(*Call actual FBs*)
fb_Move_ABS[Axis_Index](Axis:= Axis[Axis_Index]);
IF ReadyFor_Motion[Axis_Index] AND In_Play_ACK[Axis_Index] AND NOT FB_In.Stop_PlayBack[Axis_Index] AND NOT Cycle_Complete[Axis_Index]
	THEN
			(*---------------Explicit Step Call-------------*)
			IF (FB_In.Start_Explicit_StepCall[Axis_Index] OR Step_Running[Axis_Index])
				AND (NOT FB_In.Start_PlayBack[Axis_Index] OR Step_Running[Axis_Index]) AND NOT Program_Running[Axis_Index]
				AND NOT Step_Complete[Axis_Index]
				AND (Current_Step_Pointer[Axis_Index]>=1) AND (Current_Step_Pointer[Axis_Index]<=15)
					THEN
					Step_Running[Axis_Index]:= TRUE;
					Current_Step_Pointer[Axis_Index]:= FB_In.Explicit_Step_REQ[Axis_Index];
					(*--- Absolute Type Move Requested ---*)
					IF NOT fb_Move_ABS[Axis_Index].Active AND NOT fb_Move_Vel[Axis_Index].Active AND NOT fb_Move_MOD[Axis_Index].Active
						AND NOT fb_Move_ABS[Axis_Index].Execute AND NOT fb_Move_Vel[Axis_Index].Execute AND NOT fb_Move_MOD[Axis_Index].Execute
						AND (Program_Positions[Axis_Index][Current_Step_Pointer[Axis_Index]].Move_Type=0)
						THEN
						(*Set Auto Playback Parameters Per Position*)
						fb_Move_ABS[Axis_Index].Velocity:= (Program_Positions[Axis_Index] [Current_Step_Pointer[Axis_Index]].Velocity *(FB_In.PlayBack_Speed_Percentage[Axis_Index]/100));
						fb_Move_ABS[Axis_Index].Acceleration:= Program_Positions[Axis_Index][Current_Step_Pointer[Axis_Index]].Accel;
						fb_Move_ABS[Axis_Index].Deceleration:= Program_Positions[Axis_Index][Current_Step_Pointer[Axis_Index]].Decel;
						fb_Move_ABS[Axis_Index].Position:= Program_Positions[Axis_Index][Current_Step_Pointer[Axis_Index]].Position;
						fb_Move_ABS[Axis_Index].Execute:= TRUE;
					ELSIF fb_Move_ABS[Axis_Index].Execute AND fb_Move_ABS[Axis_Index].Done AND In_Requested_Position[Axis_Index] AND (At_Current_Step[Axis_Index] = Current_Step_Pointer[Axis_Index])
						THEN
							fb_Move_ABS[Axis_Index].Execute:= FALSE;			(*Position Reached, step execution request*)
							Step_Complete[Axis_Index]:= TRUE;
					END_IF;

			END_IF;

			(*--------------Cycle through Programmed Steps Continuous until End-----------*)
			IF (FB_In.Start_PlayBack[Axis_Index])
				AND fb_Power[Axis_Index].Status (*MC_Power -> Status:=Control Loop Closed (new ready bit (StateDWord.20) and not in error*)
				AND NOT FB_In.Start_Explicit_StepCall[Axis_Index] AND NOT Step_Running[Axis_Index]
				AND NOT Program_Complete[Axis_Index] AND FB_In.PlayBack_StepPermit[Axis_Index]
				AND ((NOT Program_Running[Axis_Index] AND ((Current_Step_Pointer[Axis_Index]=1) AND In_Requested_Position[Axis_Index]))
				OR (Program_Running[Axis_Index] AND (Current_Step_Pointer[Axis_Index]>=1) AND (Current_Step_Pointer[Axis_Index]<=15)))
					THEN
					Program_Running[Axis_Index]:= TRUE;
					IF NOT fb_Move_ABS[Axis_Index].Active AND NOT fb_Move_ABS[Axis_Index].Execute
						AND NOT fb_Move_MOD[Axis_Index].Active AND NOT fb_Move_MOD[Axis_Index].Execute
						AND (Program_Positions[Axis_Index][Current_Step_Pointer[Axis_Index]].Move_Type=0)
						THEN
						(*Set Auto Playback Parameters Per Position*)
						fb_Move_ABS[Axis_Index].Velocity:= (Program_Positions[Axis_Index][Current_Step_Pointer[Axis_Index]].Velocity *(FB_In.PlayBack_Speed_Percentage[Axis_Index]/100));
						fb_Move_ABS[Axis_Index].Acceleration:= Program_Positions[Axis_Index][Current_Step_Pointer[Axis_Index]].Accel;
						fb_Move_ABS[Axis_Index].Deceleration:= Program_Positions[Axis_Index][Current_Step_Pointer[Axis_Index]].Decel;
						fb_Move_ABS[Axis_Index].Position:= Program_Positions[Axis_Index][Current_Step_Pointer[Axis_Index]].Position;
						fb_Move_ABS[Axis_Index].Execute:= TRUE;
					ELSIF fb_Move_ABS[Axis_Index].Execute AND fb_Move_ABS[Axis_Index].Done AND In_Requested_Position[Axis_Index] AND (At_Current_Step[Axis_Index] = Current_Step_Pointer[Axis_Index])
						THEN
							fb_Move_ABS[Axis_Index].Execute:= FALSE; 				(*Position Reached, step execution request*)
							(*Set Program Complete Flag to Only Allow One Cycle*)
							IF Program_Running[Axis_Index] AND Current_Step_Pointer[Axis_Index]> 15 OR (Program_Positions[Axis_Index][Current_Step_Pointer[Axis_Index]].End_Flag=TRUE)
								THEN
									Program_Complete[Axis_Index]:= TRUE;
							END_IF;
							Current_Step_Pointer[Axis_Index]:= Current_Step_Pointer[Axis_Index]+1;	(*Once Position is reached, increment step pointer*)
					END_IF;
			END_IF;

(*Call actual FBs*)
fb_Move_ABS[Axis_Index](Axis:= Axis[Axis_Index]);

				(*Reset Complete Flag and Step Pointer*)
				IF (Program_Complete[Axis_Index] AND Program_Running[Axis_Index]) OR FB_In.Program_Reset[Axis_Index]
					THEN
						Current_Step_Pointer[Axis_Index]:= 1;
						IF NOT fb_Move_ABS[Axis_Index].Busy AND NOT fb_Move_ABS[Axis_Index].Execute
							AND NOT fb_Move_MOD[Axis_Index].Busy AND NOT fb_Move_MOD[Axis_Index].Execute
							THEN
							(*Set Auto Playback Parameters Per Position*)
							fb_Move_ABS[Axis_Index].Velocity:= (Program_Positions[Axis_Index][Current_Step_Pointer[Axis_Index]].Velocity *(FB_In.PlayBack_Speed_Percentage[Axis_Index]/100));
							fb_Move_ABS[Axis_Index].Acceleration:= Program_Positions[Axis_Index][Current_Step_Pointer[Axis_Index]].Accel;
							fb_Move_ABS[Axis_Index].Deceleration:= Program_Positions[Axis_Index][Current_Step_Pointer[Axis_Index]].Decel;
							fb_Move_ABS[Axis_Index].Position:= Program_Positions[Axis_Index][Current_Step_Pointer[Axis_Index]].Position;
							fb_Move_ABS[Axis_Index].Execute:= TRUE;
						ELSIF fb_Move_ABS[Axis_Index].Execute AND fb_Move_ABS[Axis_Index].Done AND In_Requested_Position[Axis_Index] AND (At_Current_Step[Axis_Index] = Current_Step_Pointer[Axis_Index])
							THEN
								fb_Move_ABS[Axis_Index].Execute:= FALSE; 				(*Position Reached, step execution request*)
								Program_Complete[Axis_Index]:= FALSE;
								Program_Running[Axis_Index]:= FALSE;
								Cycle_Complete[Axis_Index]:= TRUE;
						END_IF;
				END_IF;



ELSE
	fb_Move_ABS[Axis_Index].Execute:= FALSE;
	fb_Move_VEL[Axis_Index].Execute:= FALSE;
	fb_Move_MOD[Axis_Index].Execute:= FALSE;
	Step_Complete[Axis_Index]:= FALSE;
	Step_Running[Axis_Index]:= FALSE;

END_IF; (*End_If for Play Loop*)
END_ACTION

ACTION Move_Modulo:
(*General Set-Up Parameters/Function calls for Servo Drive*)

(*Call actual FBs*)
fb_Move_MOD[Axis_Index](Axis:= Axis[Axis_Index]);
IF ReadyFor_Motion[Axis_Index] AND In_Play_ACK[Axis_Index] AND NOT FB_In.Stop_PlayBack[Axis_Index] AND NOT Cycle_Complete[Axis_Index]
	THEN
			(*---------------Explicit Step Call-------------*)
			IF (FB_In.Start_Explicit_StepCall[Axis_Index] OR Step_Running[Axis_Index])
				AND (NOT FB_In.Start_PlayBack[Axis_Index] OR Step_Running[Axis_Index]) AND NOT Program_Running[Axis_Index]
				AND NOT Step_Complete[Axis_Index]
				AND (Current_Step_Pointer[Axis_Index]>=1) AND (Current_Step_Pointer[Axis_Index]<=15)
					THEN
					Step_Running[Axis_Index]:= TRUE;
					Current_Step_Pointer[Axis_Index]:= FB_In.Explicit_Step_REQ[Axis_Index];
					(*--- Modulo Type Move Requested ---*)
					IF NOT fb_Move_ABS[Axis_Index].Active AND NOT fb_Move_Vel[Axis_Index].Active AND NOT fb_Move_MOD[Axis_Index].Active
						AND NOT fb_Move_ABS[Axis_Index].Execute AND NOT fb_Move_Vel[Axis_Index].Execute AND NOT fb_Move_MOD[Axis_Index].Execute
						AND (Program_Positions[Axis_Index][Current_Step_Pointer[Axis_Index]].Move_Type=3)
						THEN
						(*Set Auto Playback Parameters Per Position*)
						fb_Move_MOD[Axis_Index].Velocity:= (Program_Positions[Axis_Index] [Current_Step_Pointer[Axis_Index]].Velocity *(FB_In.PlayBack_Speed_Percentage[Axis_Index]/100));
						fb_Move_MOD[Axis_Index].Acceleration:= Program_Positions[Axis_Index][Current_Step_Pointer[Axis_Index]].Accel;
						fb_Move_MOD[Axis_Index].Deceleration:= Program_Positions[Axis_Index][Current_Step_Pointer[Axis_Index]].Decel;
						fb_Move_MOD[Axis_Index].Position:= Program_Positions[Axis_Index][Current_Step_Pointer[Axis_Index]].Position;
						fb_Move_MOD[Axis_Index].Execute:= TRUE;
					ELSIF fb_Move_MOD[Axis_Index].Execute AND fb_Move_MOD[Axis_Index].Done AND In_Requested_Position[Axis_Index] AND (At_Current_Step[Axis_Index] = Current_Step_Pointer[Axis_Index])
						THEN
							fb_Move_MOD[Axis_Index].Execute:= FALSE;			(*Position Reached, step execution request*)
							Step_Complete[Axis_Index]:= TRUE;
					END_IF;

			END_IF;

			(*--------------Cycle through Programmed Steps Continuous until End-----------*)
			IF (FB_In.Start_PlayBack[Axis_Index])
				AND fb_Power[Axis_Index].Status (*MC_Power -> Status:=Control Loop Closed (new ready bit (StateDWord.20) and not in error*)
				AND NOT FB_In.Start_Explicit_StepCall[Axis_Index] AND NOT Step_Running[Axis_Index]
				AND NOT Program_Complete[Axis_Index] AND FB_In.PlayBack_StepPermit[Axis_Index]
				AND ((NOT Program_Running[Axis_Index] AND ((Current_Step_Pointer[Axis_Index]=1) AND In_Requested_Position[Axis_Index]))
				OR (Program_Running[Axis_Index] AND (Current_Step_Pointer[Axis_Index]>=1) AND (Current_Step_Pointer[Axis_Index]<=15)))
					THEN
					Program_Running[Axis_Index]:= TRUE;
					IF NOT fb_Move_ABS[Axis_Index].Active AND NOT fb_Move_ABS[Axis_Index].Execute
						AND NOT fb_Move_MOD[Axis_Index].Active AND NOT fb_Move_MOD[Axis_Index].Execute
						AND (Program_Positions[Axis_Index][Current_Step_Pointer[Axis_Index]].Move_Type=0)
						THEN
						(*Set Auto Playback Parameters Per Position*)
						fb_Move_MOD[Axis_Index].Velocity:= (Program_Positions[Axis_Index][Current_Step_Pointer[Axis_Index]].Velocity *(FB_In.PlayBack_Speed_Percentage[Axis_Index]/100));
						fb_Move_MOD[Axis_Index].Acceleration:= Program_Positions[Axis_Index][Current_Step_Pointer[Axis_Index]].Accel;
						fb_Move_MOD[Axis_Index].Deceleration:= Program_Positions[Axis_Index][Current_Step_Pointer[Axis_Index]].Decel;
						fb_Move_MOD[Axis_Index].Position:= Program_Positions[Axis_Index][Current_Step_Pointer[Axis_Index]].Position;
						fb_Move_MOD[Axis_Index].Execute:= TRUE;
					ELSIF fb_Move_MOD[Axis_Index].Execute AND fb_Move_MOD[Axis_Index].Done AND In_Requested_Position[Axis_Index] AND (At_Current_Step[Axis_Index] = Current_Step_Pointer[Axis_Index])
						THEN
							fb_Move_MOD[Axis_Index].Execute:= FALSE; 				(*Position Reached, step execution request*)
							(*Set Program Complete Flag to Only Allow One Cycle*)
							IF Program_Running[Axis_Index] AND Current_Step_Pointer[Axis_Index]> 15 OR (Program_Positions[Axis_Index][Current_Step_Pointer[Axis_Index]].End_Flag=TRUE)
								THEN
									Program_Complete[Axis_Index]:= TRUE;
							END_IF;
							Current_Step_Pointer[Axis_Index]:= Current_Step_Pointer[Axis_Index]+1;	(*Once Position is reached, increment step pointer*)
					END_IF;
			END_IF;

(*Call actual FBs*)
fb_Move_MOD[Axis_Index](Axis:= Axis[Axis_Index]);

				(*Reset Complete Flag and Step Pointer*)
				IF (Program_Complete[Axis_Index] AND Program_Running[Axis_Index]) OR FB_In.Program_Reset[Axis_Index]
					THEN
						Current_Step_Pointer[Axis_Index]:= 1;
						IF NOT fb_Move_ABS[Axis_Index].Busy AND NOT fb_Move_ABS[Axis_Index].Execute
							AND NOT fb_Move_MOD[Axis_Index].Busy AND NOT fb_Move_MOD[Axis_Index].Execute
							THEN
							(*Set Auto Playback Parameters Per Position*)
							fb_Move_MOD[Axis_Index].Velocity:= (Program_Positions[Axis_Index][Current_Step_Pointer[Axis_Index]].Velocity *(FB_In.PlayBack_Speed_Percentage[Axis_Index]/100));
							fb_Move_MOD[Axis_Index].Acceleration:= Program_Positions[Axis_Index][Current_Step_Pointer[Axis_Index]].Accel;
							fb_Move_MOD[Axis_Index].Deceleration:= Program_Positions[Axis_Index][Current_Step_Pointer[Axis_Index]].Decel;
							fb_Move_MOD[Axis_Index].Position:= Program_Positions[Axis_Index][Current_Step_Pointer[Axis_Index]].Position;
							fb_Move_MOD[Axis_Index].Execute:= TRUE;
						ELSIF fb_Move_MOD[Axis_Index].Execute AND fb_Move_MOD[Axis_Index].Done AND In_Requested_Position[Axis_Index] AND (At_Current_Step[Axis_Index] = Current_Step_Pointer[Axis_Index])
							THEN
								fb_Move_MOD[Axis_Index].Execute:= FALSE; 				(*Position Reached, step execution request*)
								Program_Complete[Axis_Index]:= FALSE;
								Program_Running[Axis_Index]:= FALSE;
								Cycle_Complete[Axis_Index]:= TRUE;
						END_IF;
				END_IF;



ELSE
	fb_Move_ABS[Axis_Index].Execute:= FALSE;
	fb_Move_VEL[Axis_Index].Execute:= FALSE;
	fb_Move_MOD[Axis_Index].Execute:= FALSE;
	Step_Complete[Axis_Index]:= FALSE;
	Step_Running[Axis_Index]:= FALSE;

END_IF; (*End_If for Play Loop*)
END_ACTION

ACTION Move_Velocity:
(*General Set-Up Parameters/Function calls for Servo Drive*)

(*Call actual FBs*)
fb_Move_Vel[Axis_Index](Axis:= Axis[Axis_Index]);

IF ReadyFor_Motion[Axis_Index] AND In_Play_ACK[Axis_Index] AND NOT FB_In.Stop_PlayBack[Axis_Index] AND NOT Cycle_Complete[Axis_Index]
	THEN
			(*---------------Explicit Step Call-------------*)
			IF (FB_In.Start_Explicit_StepCall[Axis_Index] OR Step_Running[Axis_Index])
				AND (NOT FB_In.Start_PlayBack[Axis_Index] OR Step_Running[Axis_Index]) AND NOT Program_Running[Axis_Index]
				AND NOT Step_Complete[Axis_Index]
				AND (Current_Step_Pointer[Axis_Index]>=1) AND (Current_Step_Pointer[Axis_Index]<=15)
					THEN
					Step_Running[Axis_Index]:= TRUE;
					Current_Step_Pointer[Axis_Index]:= FB_In.Explicit_Step_REQ[Axis_Index];

					(*--- Velocity only type move requested (+ or - direction) ---*)
					IF NOT fb_Move_ABS[Axis_Index].Active AND NOT fb_Move_Vel[Axis_Index].Active AND NOT fb_Move_MOD[Axis_Index].Active
						AND NOT fb_Move_ABS[Axis_Index].Execute AND NOT fb_Move_Vel[Axis_Index].Execute AND NOT fb_Move_MOD[Axis_Index].Execute
						AND ((Program_Positions[Axis_Index][Current_Step_Pointer[Axis_Index]].Move_Type=1) OR  (Program_Positions[Axis_Index][Current_Step_Pointer[Axis_Index]].Move_Type=2))

						THEN
						(*Set Auto Playback Parameters Per Position*)
						fb_Move_VEL[Axis_Index].Velocity:= (Program_Positions[Axis_Index] [Current_Step_Pointer[Axis_Index]].Velocity *(FB_In.PlayBack_Speed_Percentage[Axis_Index]/100));
						fb_Move_VEL[Axis_Index].Acceleration:= Program_Positions[Axis_Index][Current_Step_Pointer[Axis_Index]].Accel;
						fb_Move_VEL[Axis_Index].Deceleration:= Program_Positions[Axis_Index][Current_Step_Pointer[Axis_Index]].Decel;
						(*Set Directionality*)
						IF (Program_Positions[Axis_Index][Current_Step_Pointer[Axis_Index]].Move_Type=1) (*+ direction requested*)
							THEN
							fb_Move_VEL[Axis_Index].Direction:= MC_Positive_Direction; (*Set Direction to Positive*)
						ELSIF (Program_Positions[Axis_Index][Current_Step_Pointer[Axis_Index]].Move_Type=2) (*- direction requested*)
							THEN
							fb_Move_VEL[Axis_Index].Direction:= MC_Negative_Direction; (*Set Direction to Positive*)
						END_IF;
						fb_Move_VEL[Axis_Index].Execute:= TRUE;
					END_IF;
			END_IF;

ELSE
	fb_Move_ABS[Axis_Index].Execute:= FALSE;
	fb_Move_VEL[Axis_Index].Execute:= FALSE;
	fb_Move_MOD[Axis_Index].Execute:= FALSE;
	Step_Complete[Axis_Index]:= FALSE;
	Step_Running[Axis_Index]:= FALSE;

END_IF; (*End_If for Play Loop*)
END_ACTION

ACTION Teach_Mode:
(*################################################# Manual Mode Code ###########################################*)
(*General Set-Up Parameters/Function calls for Servo Drive*)
			fb_Jog[Axis_Index](Axis:= Axis[Axis_Index]);
			fb_Move_ABSTeach[Axis_Index](Axis:= Axis[Axis_Index]);
			fb_Set_Home[Axis_Index](Axis:= Axis[Axis_Index]);
			SET_HomeTMR[Axis_Index].PT:= T#5.0s;							(*Preset Time for Teach HomePos*)

IF ReadyFor_TeachMotion[Axis_Index] AND In_Teach_ACK[Axis_Index] AND NOT fb_Stop[Axis_Index].Execute
	THEN
		Current_Step_Pointer[Axis_Index]:= FB_In.Explicit_Step_REQ[Axis_Index];
		Step_Complete[Axis_Index]:= FALSE;
		Step_Running[Axis_Index]:= FALSE;
		Program_Complete[Axis_Index]:= FALSE;
		Program_Running[Axis_Index]:= FALSE;

			(*---------------Explicit Step Call in Teach-------------*)
			IF FB_In.Start_Explicit_StepCall[Axis_Index] AND ReadyFor_Motion[Axis_Index]
				AND (Current_Step_Pointer[Axis_Index]>=1) AND (Current_Step_Pointer[Axis_Index]<=15)
					THEN
					(*--- Absolute Type Move Requested ---*)
					IF NOT fb_Move_ABS[Axis_Index].Active AND NOT fb_Move_Vel[Axis_Index].Active AND NOT fb_Move_MOD[Axis_Index].Active
						AND NOT fb_Move_ABS[Axis_Index].Execute AND NOT fb_Move_Vel[Axis_Index].Execute AND NOT fb_Move_MOD[Axis_Index].Execute
						AND (Program_Positions[Axis_Index][Current_Step_Pointer[Axis_Index]].Move_Type=0)
						THEN
						(*Set Auto Playback Parameters Per Position*)
						fb_Move_ABS[Axis_Index].Velocity:= 250; (*In Teach Mode, Lock down Velcoity*)
						fb_Move_ABS[Axis_Index].Acceleration:= Program_Positions[Axis_Index][Current_Step_Pointer[Axis_Index]].Accel;
						fb_Move_ABS[Axis_Index].Deceleration:= Program_Positions[Axis_Index][Current_Step_Pointer[Axis_Index]].Decel;
						fb_Move_ABS[Axis_Index].Position:= Program_Positions[Axis_Index][Current_Step_Pointer[Axis_Index]].Position;
						fb_Move_ABS[Axis_Index].Execute:= TRUE;
					ELSIF fb_Move_ABS[Axis_Index].Execute AND fb_Move_ABS[Axis_Index].Done AND In_Requested_Position[Axis_Index] AND (At_Current_Step[Axis_Index] = Current_Step_Pointer[Axis_Index])
						THEN
							fb_Move_ABS[Axis_Index].Execute:= FALSE;			(*Position Reached, step execution request*)
					END_IF;
					(*--- Modulo Type Move Requested ---*)
					IF NOT fb_Move_ABS[Axis_Index].Active AND NOT fb_Move_Vel[Axis_Index].Active AND NOT fb_Move_MOD[Axis_Index].Active
						AND NOT fb_Move_ABS[Axis_Index].Execute AND NOT fb_Move_Vel[Axis_Index].Execute AND NOT fb_Move_MOD[Axis_Index].Execute
						AND (Program_Positions[Axis_Index][Current_Step_Pointer[Axis_Index]].Move_Type=3)
						THEN
						(*Set Auto Playback Parameters Per Position*)
						fb_Move_MOD[Axis_Index].Velocity:= 250; (*In Teach Mode, Lock down Velcoity*)
						fb_Move_MOD[Axis_Index].Acceleration:= Program_Positions[Axis_Index][Current_Step_Pointer[Axis_Index]].Accel;
						fb_Move_MOD[Axis_Index].Deceleration:= Program_Positions[Axis_Index][Current_Step_Pointer[Axis_Index]].Decel;
						fb_Move_MOD[Axis_Index].Position:= Program_Positions[Axis_Index][Current_Step_Pointer[Axis_Index]].Position;
						fb_Move_MOD[Axis_Index].Execute:= TRUE;
					ELSIF fb_Move_MOD[Axis_Index].Execute AND fb_Move_MOD[Axis_Index].Done AND In_Requested_Position[Axis_Index] AND (At_Current_Step[Axis_Index] = Current_Step_Pointer[Axis_Index])
						THEN
							fb_Move_MOD[Axis_Index].Execute:= FALSE;			(*Position Reached, step execution request*)
					END_IF;
					(*--- Velocity only type move requested (+ or - direction) ---*)
					IF NOT fb_Move_ABS[Axis_Index].Active AND NOT fb_Move_Vel[Axis_Index].Active
						AND NOT fb_Move_ABS[Axis_Index].Execute AND NOT fb_Move_Vel[Axis_Index].Execute
						AND ((Program_Positions[Axis_Index][Current_Step_Pointer[Axis_Index]].Move_Type=1) OR  (Program_Positions[Axis_Index][Current_Step_Pointer[Axis_Index]].Move_Type=2))
						THEN
						(*Set Auto Playback Parameters Per Position*)
						fb_Move_VEL[Axis_Index].Velocity:= 250; (*In Teach Mode, Lock down Velcoity*)
						fb_Move_VEL[Axis_Index].Acceleration:= Program_Positions[Axis_Index][Current_Step_Pointer[Axis_Index]].Accel;
						fb_Move_VEL[Axis_Index].Deceleration:= Program_Positions[Axis_Index][Current_Step_Pointer[Axis_Index]].Decel;
						(*Set Directionality*)
						IF (Program_Positions[Axis_Index][Current_Step_Pointer[Axis_Index]].Move_Type=1) (*+ direction requested*)
							THEN
							fb_Move_VEL[Axis_Index].Direction:= MC_Positive_Direction; (*Set Direction to Positive*)
						ELSIF (Program_Positions[Axis_Index][Current_Step_Pointer[Axis_Index]].Move_Type=2) (*- direction requested*)
							THEN
							fb_Move_VEL[Axis_Index].Direction:= MC_Negative_Direction; (*Set Direction to Positive*)
						END_IF;
						fb_Move_VEL[Axis_Index].Execute:= TRUE;
					END_IF;
			ELSE
				fb_Move_ABS[Axis_Index].Execute:= FALSE;
				fb_Move_VEL[Axis_Index].Execute:= FALSE;
				fb_Move_MOD[Axis_Index].Execute:= FALSE;
			END_IF;
(*Call actual FBs*)
fb_Move_ABS[Axis_Index](Axis:= Axis[Axis_Index]);
fb_Move_Vel[Axis_Index](Axis:= Axis[Axis_Index]);
fb_Move_MOD[Axis_Index](Axis:= Axis[Axis_Index]);
			(*Set Inching Value*)
			IF FB_In.Teach_MicroInch_Enable[Axis_Index]
				THEN
				Inching_Value[Axis_Index]:= FB_In.MicroInch_Value[Axis_Index];
			ELSE
				Inching_Value[Axis_Index]:= 0.5;	(*Default Inching Value is 0.5mm OR degrees (depending on how Motion System is config'd*)
			END_IF;
			(*-------------Jog and Inching -----------------------*)
			IF FB_In.Teach_JogFast_Plus[Axis_Index] OR FB_In.Teach_JogFast_Minus[Axis_Index]
				THEN
					(*Jog Drive Fast*)
					fb_Jog[Axis_Index].Mode:= MC_JOGMODE_STANDARD_FAST;
					fb_Jog[Axis_Index].Acceleration:= 0;
					fb_Jog[Axis_Index].Velocity:= 0;
					fb_Jog[Axis_Index].JogForward:= FB_In.Teach_JogFast_Plus[Axis_Index];
					fb_Jog[Axis_Index].JogBackwards:= FB_In.Teach_JogFast_Minus[Axis_Index];
			ELSIF FB_In.Teach_JogSlow_Plus[Axis_Index] OR FB_In.Teach_JogSlow_Minus[Axis_Index]
				THEN
					(*Jog Drive Slow*)
					fb_Jog[Axis_Index].Mode:= MC_JOGMODE_STANDARD_SLOW;
					fb_Jog[Axis_Index].Acceleration:= 0;
					fb_Jog[Axis_Index].Velocity:= 0;
					fb_Jog[Axis_Index].JogForward:= FB_In.Teach_JogSlow_Plus[Axis_Index];
					fb_Jog[Axis_Index].JogBackwards:= FB_In.Teach_JogSlow_Minus[Axis_Index];
			ELSIF FB_In.Teach_Inch_Plus[Axis_Index] OR FB_In.Teach_Inch_Minus[Axis_Index]
				THEN
					(*Jog Drive Inching*)
					fb_Jog[Axis_Index].Mode:= MC_JOGMODE_INCHING;
					fb_Jog[Axis_Index].Position:= Inching_Value[Axis_Index];
					fb_Jog[Axis_Index].Acceleration:= 10;
					fb_Jog[Axis_Index].Velocity:= 10;
					fb_Jog[Axis_Index].JogForward:= FB_In.Teach_Inch_Plus[Axis_Index];
					fb_Jog[Axis_Index].JogBackwards:= FB_In.Teach_Inch_Minus[Axis_Index];
			ELSE
					fb_Jog[Axis_Index].JogForward:= FALSE;
					fb_Jog[Axis_Index].JogBackwards:= FALSE;
			END_IF; (*End_If for Jog/Inch Requests*)

			(*---------------- Record Current Position -----------------*)
			IF ReadyFor_Motion[Axis_Index] AND FB_In.Teach_Record_CurrentPos[Axis_Index] AND FB_in.Teach_Enable[Axis_Index]
				THEN
				IF FB_In.Teach_Params[Axis_Index].Move_Type=0 (*Abs Move Type*)
					THEN
					IF (FB_In.Teach_Params[Axis_Index].Velocity=0) AND (FB_In.Teach_Params[Axis_Index].Accel=0)
						AND (FB_In.Teach_Params[Axis_Index].Decel=0) AND (FB_In.Teach_Params[Axis_Index].Move_Type=0)
						AND (FB_In.Teach_Params[Axis_Index].End_Flag=0) AND FB_In.Teach_ParamsOverwrite_Flag[Axis_Index]
						THEN
						Program_Positions[Axis_Index][Current_Step_Pointer[Axis_Index]].Position:= 0; 									(*If All input paramters are set to zero and overwrite is selected then user is requesting to blank step*)
					ELSIF  (FB_In.Teach_Params[Axis_Index].Velocity>0)
						THEN
						Program_Positions[Axis_Index][Current_Step_Pointer[Axis_Index]].Position:= Current_Position[Axis_Index];				(*Store Current Positional Data to Program at Current Pointer Location*)
					END_IF;
				ELSIF FB_In.Teach_Params[Axis_Index].Move_Type=1 OR FB_In.Teach_Params[Axis_Index].Move_Type=2 (*Vel Move Type + or - *)
					THEN
					Program_Positions[Axis_Index][Current_Step_Pointer[Axis_Index]].Position:= 0; 														(*If Move Type is Velocity only, then blank Positional data*)
				END_IF;
				(*Only overwrite all other parameters if Overwirte is selected*)
				IF FB_In.Teach_ParamsOverwrite_Flag[Axis_Index]
					THEN
					Program_Positions[Axis_Index][Current_Step_Pointer[Axis_Index]].Velocity:= (FB_In.System_Max_Velocity[Axis_Index] *(FB_In.Teach_Params[Axis_Index].Velocity/100)); 	(*Servo System Maximum Velocity x Desired PlayBack Speed*)
					Program_Positions[Axis_Index][Current_Step_Pointer[Axis_Index]].Accel:= FB_In.Teach_Params[Axis_Index].Accel;												(*Store Accel Param*)
					Program_Positions[Axis_Index][Current_Step_Pointer[Axis_Index]].Decel:= FB_In.Teach_Params[Axis_Index].Decel;												(*Store Decel Param*)
					Program_Positions[Axis_Index][Current_Step_Pointer[Axis_Index]].Move_Type:= FB_In.Teach_Params[Axis_Index].Move_Type;									(*Store Decel Param*)
					Program_Positions[Axis_Index][Current_Step_Pointer[Axis_Index]].End_Flag:= FB_In.Teach_Params[Axis_Index].End_Flag;										(*Store End Flag Param*)
				END_IF;
			END_IF;

			(*--------------- Set Home Routine -----------------------*)
			(*Simple Direct, Delayed Homing Routine*)
			SET_HomeTMR[Axis_Index].IN:= FB_In.Enable_Motion[Axis_Index] AND
											FB_In.Teach_Servo_HomePos[Axis_Index] AND
											FB_In.Home_Position_Switch[Axis_Index] AND NOT
											FB_In.Quick_Home_REQ[Axis_Index];
			SET_HomeTMR[Axis_Index]();

			(*User Specified, Non-Delayed Homing Routine*)
			RPulse[0].CLK:= FB_In.Enable_Motion[Axis_Index] AND
							FB_In.Quick_Home_REQ[Axis_Index] AND NOT
							FB_In.Teach_Servo_HomePos[Axis_Index] AND NOT
							SET_HomeTMR[Axis_Index].Q AND NOT
							Homed[Axis_Index];
			RPulse[0]();

			IF SET_HomeTMR[Axis_Index].Q
				THEN
					fb_Set_Home[Axis_Index].HomingMode:= MC_Direct;
					fb_Set_Home[Axis_Index].Position:=0.0;
					fb_Set_Home[Axis_Index].Execute:= TRUE;
			ELSIF RPulse[0].Q OR (fb_Set_Home[Axis_Index].Busy AND NOT FB_In.Teach_Servo_HomePos[Axis_Index] AND NOT fb_Set_Home[Axis_Index].Done)
				THEN
					fb_Set_Home[Axis_Index].HomingMode:= FB_In.Homing_Type[Axis_Index];
					fb_Set_Home[Axis_Index].bCalibrationCam:= FB_In.Home_Position_Switch[Axis_Index];
					fb_Set_Home[Axis_Index].Position:=FB_In.Homing_Offset[Axis_index];
					fb_Set_Home[Axis_Index].Execute:= TRUE;
			ELSE
					fb_Set_Home[Axis_Index].Execute:= FALSE;
			END_IF;




			IF (NOT FB_In.Axis_Is_Absolute[Axis_Index] AND fb_Set_Home[Axis_Index].Done AND NOT fb_Set_Home[Axis_Index].Error)
				THEN
					Homed[Axis_Index]:= TRUE;
			END_IF;

END_IF; (*Manual Mode End_If*)
END_ACTION

END_FUNCTION_BLOCK

// ---- POUs/FBs/FB_Ax5805_GetInfo_20200609.TcPOU
(*Function Block to read the internal data and diagnostic Data of the AX5805 to assist with troubleshooting*)
(*
Authored By - Chris Timmermans of Edge Automation
Rev 1.0 - Initial Setup
------------------------------------------------------------------------------------------
REVISION NOTES:
	Version 20160803
	- Changed data type to remove dependance on external resources, b.lekx-toniolo
	- Change ADS Net Id input to match our standard Infodata type, b.lekx-toniolo

	Version 20200609
	- Added Var_Input to pass in axis count, various code changes to error handing based on this input, b.lekx-toniolo	
------------------------------------------------------------------------------------------


*)

FUNCTION_BLOCK FB_Ax5805_GetInfo_20200609
VAR_INPUT
	Ecat_Master_AmsNetID: STRING;
	AX5805_InfoData: udt_ECATSlave_StatusEXT;
	Axis_Count: UINT;		(*Axis Count Value, only 1 or 2 is Valid*)

END_VAR
VAR_OUTPUT
	bError:	BOOL;
	bReadError: BOOL;
	bAxisCountError: BOOL;
	Data:	udt_AX5805_DiagData;
END_VAR
VAR
	Timer:				TON;
	fbCoERead_IntData1:				FB_EcCoESdoRead;
	fbCoERead_IntData2:				FB_EcCoESdoRead;
	fbCoERead_DiagData1:			FB_EcCoESdoRead;
	fbCoERead_DiagData2:			FB_EcCoESdoRead;



END_VAR

(*CoE Read uses EtherCAT service Mail box, reading of objects is scheduled to prevent overload*)

(*Pulse Timer setup - Pulse Stays true for one scan and then resets*)
Timer.PT:=T#1s;
Timer.IN:=TRUE;


IF Timer.Q THEN
	Timer.IN:=FALSE;
END_IF
Timer();

(*Read of CoE Objects*)
(*Read the internal data of the AX5805 to determine STO reason Code*)

IF Axis_Count = 1 THEN
	(*Single Axis Type Drive*)
	fbCoERead_IntData1(
		sNetId:= Ecat_Master_AmsNetID,
		nSlaveAddr:= AX5805_InfoData.AdsAddr.port ,
		nSubIndex:= 7,
		nIndex:= 16#FA10,
		pDstBuf:=ADR(Data.InternalDataA1) ,
		cbBufLen:= SIZEOF(Data.InternalDataA1),
		bExecute:= Timer.Q ,
		tTimeout:= DEFAULT_ADS_TIMEOUT,
		bBusy=> ,
		bError=> ,
		nErrId=> );

	fbCoERead_DiagData1(
		sNetId:= Ecat_Master_AmsNetID,
		nSlaveAddr:= AX5805_InfoData.AdsAddr.port ,
		nSubIndex:= 1,
		nIndex:= 16#FA82,
		pDstBuf:=ADR(Data.DiagDataA1) ,
		cbBufLen:= SIZEOF(Data.DiagDataA1),
		bExecute:= Timer.Q ,
		tTimeout:= DEFAULT_ADS_TIMEOUT,
		bBusy=> ,
		bError=> ,
		nErrId=> );

ELSIF Axis_Count = 2 THEN
	(*Dual Axis Type Drive*)
	fbCoERead_IntData2(
		sNetId:= Ecat_Master_AmsNetID,
		nSlaveAddr:= AX5805_InfoData.AdsAddr.port ,
		nSubIndex:= 8,
		nIndex:= 16#FA10,
		pDstBuf:=ADR(Data.InternalDataA2) ,
		cbBufLen:= SIZEOF(Data.InternalDataA2),
		bExecute:= Timer.Q ,
		tTimeout:= DEFAULT_ADS_TIMEOUT,
		bBusy=> ,
		bError=> ,
		nErrId=> );

	fbCoERead_DiagData2(
		sNetId:= Ecat_Master_AmsNetID,
		nSlaveAddr:= AX5805_InfoData.AdsAddr.port ,
		nSubIndex:= 2,
		nIndex:= 16#FA82,
		pDstBuf:=ADR(Data.DiagDataA2) ,
		cbBufLen:= SIZEOF(Data.DiagDataA2),
		bExecute:= Timer.Q ,
		tTimeout:= DEFAULT_ADS_TIMEOUT,
		bBusy=> ,
		bError=> ,
		nErrId=> );

ELSE
	(*Non-Valid Axis Count Value*)
	bAxisCountError:= TRUE;

END_IF;


(*If valid Axis Count was passed to this FB then Evaluate the read data from above*)

IF NOT bAxisCountError THEN
	(*Evaluate Status of Read*)
	IF 		fbCoERead_DiagData1.bError
		OR	fbCoERead_DiagData2.bError
		OR	fbCoERead_IntData1.bError
		OR	fbCoERead_IntData2.bError		THEN

			bReadError:=TRUE;
	ELSE
			bReadError:=FALSE;
	END_IF;

	(*Evaluate Status of Diag Data*)
	IF 		(Data.DiagDataA1<>0)
		OR	(Data.DiagDataA2<>0)
		OR	(Data.InternalDataA1<>0)
		OR	(Data.InternalDataA2<>0)
	THEN

			Data.bError:=TRUE;
	ELSE
			Data.bError:=FALSE;
	END_IF;

END_IF;

END_FUNCTION_BLOCK

// ---- POUs/FBs/Diagnose/AX5000 Diag/FB_AxisDiag_20160810.TcPOU
(*FB for reteiving Diags and performing systematic resets of Axis, Drive and SOE level errors

	Original Author: Beckhoff
------------------------------------------------------------------------------------------
REVISION NOTES:
	Version 20160810
		- Changed Naming to include date as per convention, b.lekx-toniolo
		- Moved two external dependaciy vars internal for protability, b.lekx-toniolo
		- Added a longer diag message string to allow full diagmessage display, b.lekx-toniolo
------------------------------------------------------------------------------------------
*)
FUNCTION_BLOCK FB_AxisDiag_20160810
VAR_INPUT
	IPCNetID				: T_AmsNetId; 	(* AmsNetId of the IPC *)
	Timeout				: TIME := DEFAULT_ADS_TIMEOUT;
	Reset				: BOOL;
	GetDiag				: BOOL;
	bLogDriveDiagMsgs 	: BOOL;
	bForceStateChgAfterDrvReset : BOOL;

END_VAR
VAR_IN_OUT
	Axis	 				: AXIS_REF;
	stAX5000Diag		: udt_AX5000Diag;
END_VAR
VAR_OUTPUT
	Error				: BOOL;
	AdsErrId				: UINT;
	SercosErrId			: UINT;
	ResetAct				: BOOL;
	DiagAct				: BOOL;
	Busy				: BOOL;
END_VAR
VAR
	iState				: INT;
	iSubState			: INT;
	GetDriveRef			: BOOL := TRUE;
	DriveRef				: ST_DriveRef; (* contains sNetID of EcMaster, nSlaveAddr of EcDrive, nDriveNo of EcDrive, either preset or read from NC *)
	AxisID				: UDINT;

	C1DErrorPrev			: BOOL;
	WcStateErrorPrev		: BOOL;
	AxisErrorPrev			: BOOL;
	OperationalPrev		: BOOL;
	ResetPrev			: BOOL;
	GetDiagPrev			: BOOL;

	fbSoERead			: FB_SoERead;
	fbDiagMessage 		: FB_SoEReadDiagMessage;
	fbClassXDiag			: FB_SoEReadClassXDiag;
	fbDiagNumber		: FB_SoEReadDiagNumber;
	fbDiagNumberList		: FB_SoEReadDiagNumberList;

	fbReset				: FB_SoEReset;
	fbDelay				: TON;
	fbGetSlaveState 		: FB_EcGetSlaveState;
	fbReqSlaveState 		: FB_EcReqSlaveState;
	fbNcReset 			: MC_Reset;

	fbAdsRead			: ADSREAD;
	readBuffer			: ARRAY[0..9] OF BYTE;
	Ids					: AMSNETID;

	fbFormatString		: FB_FormatString;
	DiagMsgPrev			: STRING(255);
	LogMsg				: STRING(255);
	strSoEString			: ST_SoE_String;
	I					: INT;
END_VAR
VAR CONSTANT
	NCIDXG_AXPARMS			: UDINT := 16#00004000;	(* Axis with ID: Parameter 			*)
	NCIDXO_AXP_HWAMSADDR	: UDINT := 16#00000031;
END_VAR

stAX5000Diag.bOperational	:= Axis.NcToPlc.StateDWord.0;
stAX5000Diag.bC1DError	 	:= Axis.NcToPlc.StateDWord.28;
stAX5000Diag.bWcStateError 	:= Axis.NcToPlc.StateDWord.30;
stAX5000Diag.bAxisError		:= Axis.NcToPlc.StateDWord.31;
stAX5000Diag.iAxisErrorCode	:= Axis.NcToPlc.ErrorCode;

CASE iState OF
0:	(* idle *)
	GetDriveRef 	:= (DriveRef.nSlaveAddr = 0);

	IF GetDriveRef THEN
		Busy			:= TRUE;
		Error			:= FALSE;
		AdsErrId		:= 0;
		SercosErrId		:= 0;
		iState 			:= 1;
		iSubState		:= 0;
		AxisID 			:= Axis.NcToPlc.AxisId;

	ELSIF Reset AND NOT ResetPrev THEN
		Busy			:= TRUE;
		ResetAct		:= TRUE;
		ResetPrev		:= Reset;
		Error			:= FALSE;
		AdsErrId		:= 0;
		SercosErrId		:= 0;
		iState 			:= 2;
		iSubState		:= 0;
		AxisID 			:= Axis.NcToPlc.AxisId;

	ELSIF GetDiag AND NOT GetDiagPrev OR
		(stAX5000Diag.bC1DError AND NOT C1DErrorPrev) OR (NOT stAX5000Diag.bC1DError AND C1DErrorPrev) (* rising/falling C1D *) OR
		(stAX5000Diag.bWcStateError AND NOT WcStateErrorPrev) OR (NOT stAX5000Diag.bWcStateError AND WcStateErrorPrev) (* rising/falling WcState *) OR
		(stAX5000Diag.bAxisError AND NOT AxisErrorPrev) OR (NOT stAX5000Diag.bAxisError AND AxisErrorPrev) (* rising/falling NcError *) OR
		(stAX5000Diag.bOperational AND NOT OperationalPrev) OR (NOT stAX5000Diag.bOperational AND OperationalPrev) (* rising/falling Enable *) THEN

		Busy			:= TRUE;
		DiagAct			:= TRUE;
		GetDiagPrev		:= GetDiag;
		Error			:= FALSE;
		AdsErrId		:= 0;
		SercosErrId		:= 0;
		iState 			:= 3;
		iSubState		:= 0;
		AxisID 			:= Axis.NcToPlc.AxisId;

		(* set/clear flags *)
		C1DErrorPrev		:= stAX5000Diag.bC1DError;
		WcStateErrorPrev	:= stAX5000Diag.bWcStateError;
		AxisErrorPrev		:= stAX5000Diag.bAxisError;
		OperationalPrev		:= stAX5000Diag.bOperational;

	ELSE
		ResetAct	:= FALSE;
		DiagAct		:= FALSE;
	END_IF

1:	(* get drive reference *)
	M_GetDriveRef();

2:	(* reset and state change *)
	M_Reset();

3:	(* get diag data *)
	M_GetDiagnosis();

END_CASE

(* clear latch *)
ResetPrev	:= ResetPrev AND Reset;
GetDiagPrev	:= GetDiagPrev AND GetDiag;

ACTION M_GetDiagnosis:
CASE iSubState OF
0:	fbClassXDiag(
		NetId		:= IPCNetID,
		Execute		:= TRUE,
		DiagClass 	:= 1,
		Timeout		:= DEFAULT_ADS_TIMEOUT,
		Axis		:= Axis,
	);

	IF NOT fbClassXDiag.Busy THEN
		fbClassXDiag(Execute:= FALSE,Axis := Axis);

		IF NOT fbClassXDiag.Error THEN
			stAX5000Diag.wClass1Diag	:= fbClassXDiag.ClassXDiag;
			stAX5000Diag.stClass1Diag	:= F_ConvWordToSTAX5000C1D(stAX5000Diag.wClass1Diag);
		ELSE
			Error			:= TRUE;
			AdsErrId		:= fbClassXDiag.AdsErrId;
			SercosErrId	:= fbClassXDiag.SercosErrId;
		END_IF
		iSubState	:= iSubState + 1;
	END_IF

1:	fbDiagMessage(
		NetId	:= IPCNetID,
		Execute	:= TRUE,
		Timeout	:= DEFAULT_ADS_TIMEOUT,
		Axis	:= Axis,
	);

	IF NOT fbDiagMessage.Busy THEN
		fbDiagMessage(Execute:= FALSE,Axis := Axis);

		IF NOT fbDiagMessage.Error THEN
			stAX5000Diag.strDiagMessage := LEFT(fbDiagMessage.DiagMessage.strData, fbDiagMessage.DiagMessage.iActualSize);
			stAX5000Diag.strDiagMessageFull := LEFT(fbDiagMessage.DiagMessage.strData, fbDiagMessage.DiagMessage.iActualSize); (*b.lekx-toniolo*)
		ELSE
			Error			:= TRUE;
			AdsErrId		:= fbDiagMessage.AdsErrId;
			SercosErrId	:= fbDiagMessage.SercosErrId;
		END_IF
		iSubState	:= iSubState + 1;
	END_IF

2:	fbDiagNumber(
		NetId	:= IPCNetID,
		Execute	:= TRUE,
		Timeout	:= DEFAULT_ADS_TIMEOUT,
		Axis	:= Axis,
	);

	IF NOT fbDiagNumber.Busy THEN
		fbDiagNumber(Execute:= FALSE,Axis := Axis);

		IF NOT fbDiagNumber.Error THEN
			stAX5000Diag.iDiagNumber := fbDiagNumber.DiagNumber;
		ELSE
			Error			:= TRUE;
			AdsErrId		:= fbDiagNumber.AdsErrId;
			SercosErrId	:= fbDiagNumber.SercosErrId;
		END_IF
		iSubState	:= iSubState + 1;
	END_IF

3:	fbSoERead(
		NetId	:= IPCNetID,
		Execute	:= TRUE,
		Idn		:= 135,
		Element	:=16#44,
		pDstBuf	:=ADR(stAX5000Diag.wDriveStatus),
		BufLen	:=SIZEOF(stAX5000Diag.wDriveStatus),
		Timeout	:= DEFAULT_ADS_TIMEOUT,
		Axis	:= Axis,
	);

	IF NOT fbSoERead.Busy THEN
		fbSoERead(Execute:= FALSE,Axis := Axis);
		IF NOT fbSoERead.Error THEN
			stAX5000Diag.stDriveStatus := F_ConvWordToSTAX5000DriveStatus(stAX5000Diag.wDriveStatus);
			iSubState		:= iSubState + 1;
		ELSE
			Error			:= TRUE;
			AdsErrId		:= fbSoERead.AdsErrId;
			SercosErrId	:= fbSoERead.SercosErrId;
			iSubState		:= iSubState + 2;
		END_IF
	END_IF

4:	fbSoERead(
		NetId	:= IPCNetID,
		Execute	:= TRUE,
		Idn		:= stAX5000Diag.stDriveStatus.iActOpModeParNum,
		Element	:=16#44,
		pDstBuf	:=ADR(stAX5000Diag.stDriveStatus.eActOpMode),
		BufLen	:=SIZEOF(stAX5000Diag.stDriveStatus.eActOpMode),
		Timeout	:= DEFAULT_ADS_TIMEOUT,
		Axis	:= Axis,
	);

	IF NOT fbSoERead.Busy THEN
		fbSoERead(Execute:= FALSE,Axis := Axis);
		IF NOT fbSoERead.Error THEN
			;
		ELSE
			Error			:= TRUE;
			AdsErrId		:= fbSoERead.AdsErrId;
			SercosErrId	:= fbSoERead.SercosErrId;
		END_IF
		iSubState	:= iSubState + 1;
	END_IF

5:	fbGetSlaveState(
		sNetId		:= DriveRef.sNetId,
		nSlaveAddr	:= DriveRef.nSlaveAddr,
		bExecute	:= TRUE,
		tTimeout	:= DEFAULT_ADS_TIMEOUT,
	);

	IF NOT fbGetSlaveState.bBusy THEN
		fbGetSlaveState(bExecute:= FALSE);
		IF NOT fbGetSlaveState.bError THEN
			stAX5000Diag.stEcSlaveState := fbGetSlaveState.state;
			stAX5000Diag.stEcSlaveStateBits := F_ConvSlaveStateToBits(fbGetSlaveState.state);
		ELSE
			Error			:= TRUE;
			AdsErrId		:= UDINT_TO_UINT(fbGetSlaveState.nErrId);
		END_IF

		IF stAX5000Diag.stEcSlaveStateBits.bError THEN
			IF stAX5000Diag.stEcSlaveStateBits.bPreop THEN
				(* read S21 - IDN List of Invalid operation data for CP2 (Preop->SaveOp) *)
				MEMSET(ADR(stAX5000Diag.stCPxInvParamList), 0, SIZEOF(stAX5000Diag.stCPxInvParamList));
				stAX5000Diag.bPreopToSafeOpError := TRUE;
				stAX5000Diag.bSafeOpToOpError := FALSE;
				iSubState	:= iSubState + 1;
			ELSIF stAX5000Diag.stEcSlaveStateBits.bSafeOp THEN
				(* read S22 - IDN List of Invalid operation data for CP3 (SaveOp->Op) *)
				MEMSET(ADR(stAX5000Diag.stCPxInvParamList), 0, SIZEOF(stAX5000Diag.stCPxInvParamList));
				stAX5000Diag.bPreopToSafeOpError := FALSE;
				stAX5000Diag.bSafeOpToOpError := TRUE;
				iSubState	:= iSubState + 2;
			ELSE
				(* Skip S21 + S22 *)
				MEMSET(ADR(stAX5000Diag.stCPxInvParamList), 0, SIZEOF(stAX5000Diag.stCPxInvParamList));
				stAX5000Diag.bPreopToSafeOpError := FALSE;
				stAX5000Diag.bSafeOpToOpError := FALSE;
				iSubState	:= iSubState + 3;
			END_IF
		ELSE
			(* Skip S21 + S22 *)
			MEMSET(ADR(stAX5000Diag.stCPxInvParamList), 0, SIZEOF(stAX5000Diag.stCPxInvParamList));
			stAX5000Diag.bPreopToSafeOpError := FALSE;
			stAX5000Diag.bSafeOpToOpError := FALSE;
			iSubState	:= iSubState + 3;
		END_IF
	END_IF

6:	(* read S21 - IDN List of Invalid operation data for CP2 (Preop->SaveOp) *)
	fbSoERead(
		NetId	:= IPCNetID,
		Execute	:= TRUE,
		Idn		:= 21,
		Element	:=16#40,
		pDstBuf	:=ADR(stAX5000Diag.stCPxInvParamList),
		BufLen	:=SIZEOF(stAX5000Diag.stCPxInvParamList),
		Timeout	:= DEFAULT_ADS_TIMEOUT,
		Axis	:= Axis,
	);

	IF NOT fbSoERead.Busy THEN
		fbSoERead(Execute:= FALSE,Axis := Axis);
		IF NOT fbSoERead.Error THEN
			;
		ELSE
			Error			:= TRUE;
			AdsErrId		:= fbSoERead.AdsErrId;
			SercosErrId	:= fbSoERead.SercosErrId;
		END_IF
		iSubState	:= iSubState + 2;
	END_IF

7:	(* read S22 - IDN List of Invalid operation data for CP3 (SaveOp->Op) *)
	fbSoERead(
		NetId	:= IPCNetID,
		Execute	:= TRUE,
		Idn		:= 22,
		Element	:=16#40,
		pDstBuf	:=ADR(stAX5000Diag.stCPxInvParamList),
		BufLen	:=SIZEOF(stAX5000Diag.stCPxInvParamList),
		Timeout	:= DEFAULT_ADS_TIMEOUT,
		Axis	:= Axis,
	);

	IF NOT fbSoERead.Busy THEN
		fbSoERead(Execute:= FALSE,Axis := Axis);
		IF NOT fbSoERead.Error THEN
			;
		ELSE
			Error			:= TRUE;
			AdsErrId		:= fbSoERead.AdsErrId;
			SercosErrId	:= fbSoERead.SercosErrId;
		END_IF
		iSubState	:= iSubState + 1;
	END_IF

8:	fbDiagNumberList(
		NetId			:= IPCNetID,
		Execute			:= TRUE,
		Timeout			:= DEFAULT_ADS_TIMEOUT,
		pDiagNumber		:= ADR(stAX5000Diag.stDiagNumberList),
		Size			:= SIZEOF(stAX5000Diag.stDiagNumberList),
		Axis			:= Axis,
	);

	IF NOT fbDiagNumberList.Busy THEN
		fbDiagNumberList(Execute:= FALSE,Axis := Axis);

		IF NOT fbDiagNumberList.Error THEN
			IF bLogDriveDiagMsgs THEN
				IF (stAX5000Diag.strDiagMessage <> DiagMsgPrev) AND (stAX5000Diag.stDiagNumberList.iActualSize > 0) THEN

					fbFormatString(
						sFormat := 'Axis ID: %d, DriveDiag: ',
						arg1 := F_UDINT(AxisID),
						sOut => LogMsg
					);
	
					FOR I := 0 TO MIN(29, stAX5000Diag.stDiagNumberList.iActualSize/4-1) DO
						IF (stAX5000Diag.stDiagNumberList.arrDiagNumbers[I] <> 0) THEN
							fbFormatString(
								sFormat := '%X, ',
								arg1 := F_UDINT(stAX5000Diag.stDiagNumberList.arrDiagNumbers[I])
							);
	
							LogMsg := CONCAT(LogMsg, fbFormatString.sOut);
						END_IF
					END_FOR
	
					LogMsg := CONCAT(LogMsg, 'DiagMsg: ');
					LogMsg := CONCAT(LogMsg, stAX5000Diag.strDiagMessage);
	
					(* report message *)
					ADSLOGSTR(msgCtrlMask := ADSLOG_MSGTYPE_ERROR OR ADSLOG_MSGTYPE_LOG,
						msgFmtStr := LogMsg, strArg:= '');
	
					DiagMsgPrev := stAX5000Diag.strDiagMessage;
				END_IF
			END_IF
		ELSE
			Error			:= TRUE;
			AdsErrId		:= fbDiagNumberList.AdsErrId;
			SercosErrId	:= fbDiagNumberList.SercosErrId;
		END_IF

		IF (stAX5000Diag.strMotorType = '') OR (stAX5000Diag.strDriveType = '') THEN
			iSubState	:= iSubState + 1;
		ELSE
			DiagAct	:= FALSE;
			iSubState	:= 0;
			iState		:= 0;
			Busy		:= FALSE;
		END_IF
	END_IF

9:	fbSoERead(
		NetId	:= IPCNetID,
		Execute	:= TRUE,
		Idn		:= P_0_IDN + 53,
		Element	:=16#44,
		pDstBuf	:=ADR(strSoEString),
		BufLen	:=SIZEOF(strSoEString),
		Timeout	:= DEFAULT_ADS_TIMEOUT,
		Axis	:= Axis,
	);

	IF NOT fbSoERead.Busy THEN
		fbSoERead(Execute:= FALSE,Axis := Axis);
		IF NOT fbSoERead.Error THEN
			MEMSET(ADR(stAX5000Diag.strMotorType),0,SIZEOF(stAX5000Diag.strMotorType));
			MEMCPY(ADR(stAX5000Diag.strMotorType),ADR(strSoEString.strData),MIN(SIZEOF(stAX5000Diag.strMotorType),strSoEString.iActualSize));
		ELSE
			Error			:= TRUE;
			AdsErrId		:= fbSoERead.AdsErrId;
			SercosErrId	:= fbSoERead.SercosErrId;
		END_IF
		iSubState	:= iSubState + 1;
	END_IF

10:	fbSoERead(
		NetId	:= IPCNetID,
		Execute	:= TRUE,
		Idn		:= P_0_IDN + 324,
		Element	:=16#44,
		pDstBuf	:=ADR(strSoEString),
		BufLen	:=SIZEOF(strSoEString),
		Timeout	:= DEFAULT_ADS_TIMEOUT,
		Axis	:= Axis,
	);

	IF NOT fbSoERead.Busy THEN
		fbSoERead(Execute:= FALSE,Axis := Axis);
		IF NOT fbSoERead.Error THEN
			MEMSET(ADR(stAX5000Diag.strDriveType),0,SIZEOF(stAX5000Diag.strDriveType));
			MEMCPY(ADR(stAX5000Diag.strDriveType),ADR(strSoEString.strData),MIN(SIZEOF(stAX5000Diag.strDriveType),strSoEString.iActualSize));
		ELSE
			Error			:= TRUE;
			AdsErrId		:= fbSoERead.AdsErrId;
			SercosErrId	:= fbSoERead.SercosErrId;
		END_IF
		DiagAct	:= FALSE;
		iSubState	:= 0;
		iState		:= 0;
		Busy		:= FALSE;
	END_IF


END_CASE
END_ACTION

ACTION M_GetDriveRef:
(* get reference from NC *)
fbAdsRead(
	NETID	:= IPCNetID,
	PORT	:= AMSPORT_R0_NC,
	IDXGRP	:= NCIDXG_AXPARMS + Axis.NcToPlc.AxisId,
	IDXOFFS	:= NCIDXO_AXP_HWAMSADDR,
	LEN		:= SIZEOF(readBuffer) ,
	DESTADDR:= ADR(readBuffer),
	READ	:= TRUE,
	TMOUT	:= Timeout
);

IF NOT fbAdsRead.BUSY THEN
	fbAdsRead(READ := FALSE);
	stAX5000Diag.nNCAxisID := Axis.NcToPlc.AxisId;

	IF NOT fbAdsRead.ERR THEN
		MEMCPY(ADR(Ids), ADR(readBuffer), SIZEOF(Ids)); 										(* readBuffer[0..5] *)
		MEMCPY(ADR(DriveRef.nSlaveAddr), ADR(readBuffer[6]), SIZEOF(DriveRef.nSlaveAddr));  	(* readBuffer[6..7] *)
		MEMCPY(ADR(DriveRef.nDriveNo), ADR(readBuffer[8]), SIZEOF(DriveRef.nDriveNo));  		(* readBuffer[8..9] *)

		(* create string out of byte array *)
		DriveRef.sNetId := F_CreateAmsNetId(Ids);
		GetDriveRef := FALSE;
	END_IF

	Busy	:= FALSE;
	iState	:= 0;
END_IF
END_ACTION

ACTION M_Reset:
CASE iSubState OF
0:
	IF stAX5000Diag.bWcStateError OR stAX5000Diag.bC1DError THEN
		(* ResetAmplifier *)
		iSubState := iSubState + 1;
	ELSIF stAX5000Diag.stEcSlaveStateBits.bError AND bForceStateChgAfterDrvReset THEN
		(* Clear Error *)
		iSubState := 4;
	ELSIF (NOT stAX5000Diag.bOperational) OR stAX5000Diag.bAxisError OR (stAX5000Diag.iAxisErrorCode <> 0) THEN
		(* NC Reset only *)
		iSubState := 6;
	ELSE
		(* reset not required *)
		iSubState	:= 0;
		iState		:= 0;
		Busy		:= FALSE;
		ResetAct	:= FALSE;
	END_IF

1:	(* ResetAmplifier *)
	fbReset(
		NetId	:= IPCNetID,
		Execute	:= TRUE,
		Timeout	:= DEFAULT_ADS_TIMEOUT,
		Axis	:= Axis,
	);
	IF NOT fbReset.Busy THEN
		fbReset(Execute:= FALSE, Axis:= Axis);

		IF NOT fbReset.Error THEN
			IF bLogDriveDiagMsgs THEN
				LogMsg := CONCAT('Axis ID: ', DWORD_TO_STRING(Axis.NcToPlc.AxisId));
				LogMsg := CONCAT(LogMsg, ', Drive Reset');

				(* report message *)
				ADSLOGSTR(msgCtrlMask := ADSLOG_MSGTYPE_ERROR OR ADSLOG_MSGTYPE_LOG,
					msgFmtStr := LogMsg, strArg:= '');

				DiagMsgPrev := '';
			END_IF
			iSubState	:= iSubState + 1;
		ELSE
			Error			:= TRUE;
			AdsErrId		:= fbReset.AdsErrId;
			SercosErrId	:= fbReset.SercosErrId;
			Busy			:= FALSE;
			ResetAct		:= FALSE;
			iSubState		:= 0;
			iState			:= 0;
		END_IF
	END_IF

2:	fbDelay(IN:=TRUE, PT:=t#3s);
	IF fbDelay.Q THEN
		fbDelay(IN:=FALSE);
		iSubState	:= iSubState + 1;
	END_IF

3:	fbGetSlaveState(
		sNetId		:= DriveRef.sNetId,
		nSlaveAddr	:= DriveRef.nSlaveAddr,
		bExecute	:= TRUE,
		tTimeout	:= DEFAULT_ADS_TIMEOUT,
	);

	IF NOT fbGetSlaveState.bBusy THEN
		fbGetSlaveState(bExecute:= FALSE);

		IF NOT fbGetSlaveState.bError THEN
			IF ((fbGetSlaveState.state.deviceState <> 16#08) OR ((fbGetSlaveState.state.deviceState AND 16#10) = 16#10)) AND
				bForceStateChgAfterDrvReset THEN

				iSubState	:= iSubState + 1;
			ELSIF Axis.NcToPlc.StateDWord.31 OR (Axis.NcToPlc.ErrorCode <> 0) THEN
				iSubState	:= 6;
			ELSE
				Busy		:= FALSE;
				ResetAct	:= FALSE;
				iSubState	:= 0;
				iState		:= 0;
			END_IF
		ELSE
			Error			:= TRUE;
			AdsErrId		:= UDINT_TO_UINT(fbGetSlaveState.nErrId);
			Busy			:= FALSE;
			ResetAct		:= FALSE;
			iSubState		:= 0;
			iState			:= 0;
		END_IF
	END_IF

4:	(* clear error *)
	fbReqSlaveState(
		sNetId		:= DriveRef.sNetId,
		nSlaveAddr	:= DriveRef.nSlaveAddr,
		bExecute	:= TRUE,
		tTimeout	:= DEFAULT_ADS_TIMEOUT,
		state		:= EC_DEVICE_STATE_ERROR);

	IF NOT fbReqSlaveState.bBusy THEN
		fbReqSlaveState(bExecute:= FALSE);

		IF NOT fbReqSlaveState.bError THEN
			iSubState	:= iSubState + 1;
		ELSE
			Error		:= TRUE;
			AdsErrId	:= UDINT_TO_UINT(fbReqSlaveState.nErrId);
			Busy		:= FALSE;
			ResetAct	:= FALSE;
			iSubState	:= 0;
			iState		:= 0;
		END_IF
	END_IF

5:	(* set op *)
	fbReqSlaveState(
		sNetId		:= DriveRef.sNetId,
		nSlaveAddr	:= DriveRef.nSlaveAddr,
		bExecute	:= TRUE,
		tTimeout	:= DEFAULT_ADS_TIMEOUT,
		state		:= EC_DEVICE_STATE_OP);

	IF NOT fbReqSlaveState.bBusy THEN
		fbReqSlaveState(bExecute:= FALSE);

		IF NOT fbReqSlaveState.bError THEN
			iSubState	:= iSubState + 1;
		ELSE
			Error		:= TRUE;
			AdsErrId	:= UDINT_TO_UINT(fbReqSlaveState.nErrId);
			Busy		:= FALSE;
			ResetAct	:= FALSE;
			iSubState	:= 0;
			iState		:= 0;
		END_IF
	END_IF

6:	fbNcReset(
		Execute:= TRUE,
		Axis:= Axis,
	);

	IF fbNcReset.Done OR fbNcReset.Error THEN
		IF fbNcReset.Error THEN
			Error 		:= TRUE;
			AdsErrId 	:= UDINT_TO_UINT(fbNcReset.ErrorID);
		END_IF

		iSubState	:= 0;
		iState		:= 0;
		Busy		:= FALSE;
		ResetAct	:= FALSE;
		fbNcReset(Execute:= FALSE, Axis:= Axis);
	END_IF
END_CASE
END_ACTION

END_FUNCTION_BLOCK

// ---- POUs/FUNs/FUN_GTAC_NC_Error_Messages.TcPOU
(*FUN for returning Error String Message based on NC error code

	Original Concept (as FB): BCM of Beckhoff?
	Original Author of this FUN: b.lekx-toniolo of Sodecia GTAC
------------------------------------------------------------------------------------------
REVISION NOTES:
	Version 20160811
		- original concept based on FB sent from Andy Burleigh of Beckhoff, b.lekx-toniolo
	Version 20221025
		- hard typed stGroupMessage and stErrorMessage to 255 to avoid build warning message, b.lekx-toniolo 
------------------------------------------------------------------------------------------
*)


FUNCTION FUN_GTAC_NC_Error_Messages : STRING
VAR_INPUT
	NC_Error_Code: UDINT;
END_VAR
VAR
	dwMask:	DWORD;
	stGroupMessage: STRING(255);
	stErrorMessage: STRING(255);
END_VAR

(*Calculate Group Index from Raw Error Code*)

dwMask := (NC_Error_Code/ 16#100);
(*
As of August 2016 from Beckhoff Infosys:

0x40nn = General errors
0x41nn = Channel Errors
0x42nn = Group Errors
0x43nn = Axis Errors
0x44nn = Encoder Errors
0x45nn = Controller Errors
0x46nn = Drive Errors
0x4Ann = Table Errors
0x4Bnn = NC PLC errors
0x4Cnn = Kinematic Transformation

0x8000 -> 0x8FFF: New extended NC error code range

0x81nn - 0x811F = Bode plot (diagnosis)
0x8120 - 0x8FFF = further errors
*)

(*---------------------------- Based on Above, Generate Group Message and Actual Error Message ---------------------------*)
(*General NC Errors*)
IF dwMask = 16#40 THEN
	stGroupMessage := 'General Error: ';
	IF NC_Error_Code = 16#4000 THEN
		stErrorMessage := 'Internal error';
	END_IF
	IF NC_Error_Code = 16#4001 THEN
		stErrorMessage := 'Memory error';
	END_IF
	IF NC_Error_Code = 16#4010 THEN
		stErrorMessage := 'Channel identifier not allowed';
	END_IF
	IF NC_Error_Code = 16#4011 THEN
		stErrorMessage := 'Group identifier not allowed';
	END_IF
	IF NC_Error_Code = 16#4012 THEN
		stErrorMessage := 'Axis identifier not allowed';
	END_IF
	IF NC_Error_Code = 16#4013 THEN
		stErrorMessage := 'Encoder identifier not allowed';
	END_IF
	IF NC_Error_Code = 16#4014 THEN
		stErrorMessage := 'Controller identifier not allowed';
	END_IF
	IF NC_Error_Code = 16#4015 THEN
		stErrorMessage := 'Drive identifier not allowed';
	END_IF
	IF NC_Error_Code = 16#4016 THEN
		stErrorMessage := 'Table identifier not allowed';
	END_IF
	IF NC_Error_Code = 16#4020 THEN
		stErrorMessage := 'No process image. No PLC-axis interface during creation of an axis. ';
	END_IF
	IF NC_Error_Code = 16#4021 THEN
		stErrorMessage := 'No process image. No axis-PLC interface during creation of an axis. ';
	END_IF
	IF NC_Error_Code = 16#4022 THEN
		stErrorMessage := 'No process image. No encoder-I/O interface during creation of an axis. ';
	END_IF
	IF NC_Error_Code = 16#4023 THEN
		stErrorMessage := 'No process image. No I/O-encoder interface during creation of an axis. ';
	END_IF
	IF NC_Error_Code = 16#4024 THEN
		stErrorMessage := 'No process image. No drive-I/O interface during creation of an axis. ';
	END_IF
	IF NC_Error_Code = 16#4025 THEN
		stErrorMessage := 'No process image. No I/O-drive interface during creation of an axis. ';
	END_IF
	IF NC_Error_Code = 16#4030 THEN
		stErrorMessage := 'Coupling type not allowed';
	END_IF
	IF NC_Error_Code = 16#4031 THEN
		stErrorMessage := 'Axis type not allowed';
	END_IF
	IF NC_Error_Code = 16#4040 THEN
		stErrorMessage := 'Axis is incompatible';
	END_IF
	IF NC_Error_Code = 16#4050 THEN
		stErrorMessage := 'Channel not ready for operation';
	END_IF
	IF NC_Error_Code = 16#4051 THEN
		stErrorMessage := 'Group not ready for operation';
	END_IF
	IF NC_Error_Code = 16#4052 THEN
		stErrorMessage := 'Axis not ready for operation';
	END_IF
	IF NC_Error_Code = 16#4060 THEN
		stErrorMessage := 'Channel exists';
	END_IF
	IF NC_Error_Code = 16#4061 THEN
		stErrorMessage := 'Group exists';
	END_IF
	IF NC_Error_Code = 16#4062 THEN
		stErrorMessage := 'Axis exists';
	END_IF
	IF NC_Error_Code = 16#4063 THEN
		stErrorMessage := 'Table exists';
	END_IF
	IF NC_Error_Code = 16#4070 THEN
		stErrorMessage := 'Axis index not allowed. The location within the channel specified for an axis is not allowed. ';
	END_IF
	IF NC_Error_Code = 16#4071 THEN
		stErrorMessage := 'Axis index not allowed. The location within the group specified for an axis is not allowed. ';
	END_IF
END_IF

(*Channel Errors*)
IF dwMask = 16#41 THEN
	stGroupMessage := 'Channel Error: ';
	IF NC_Error_Code = 16#4101 THEN
		stErrorMessage := 'Group index not allowed';
	END_IF
	IF NC_Error_Code = 16#4102 THEN
		stErrorMessage := 'Null pointer';
	END_IF
	IF NC_Error_Code = 16#4103 THEN
		stErrorMessage := 'No process image';
	END_IF
	IF NC_Error_Code = 16#4104 THEN
		stErrorMessage := 'M-function index not allowed';
	END_IF
	IF NC_Error_Code = 16#4105 THEN
		stErrorMessage := 'No memory';
	END_IF
	IF NC_Error_Code = 16#4106 THEN
		stErrorMessage := 'Not ready';
	END_IF
	IF NC_Error_Code = 16#4107 THEN
		stErrorMessage := 'Function/command not supported';
	END_IF
	IF NC_Error_Code = 16#4108 THEN
		stErrorMessage := 'Invalid parameter while starting';
	END_IF
	IF NC_Error_Code = 16#4109 THEN
		stErrorMessage := 'Channel function/command not executable';
	END_IF
	IF NC_Error_Code = 16#410A THEN
		stErrorMessage := 'ItpGoAhead not executable';
	END_IF
	IF NC_Error_Code = 16#4110 THEN
		stErrorMessage := 'Error opening a file';
	END_IF
	IF NC_Error_Code = 16#4111 THEN
		stErrorMessage := 'Syntax error during loading';
	END_IF
	IF NC_Error_Code = 16#4112 THEN
		stErrorMessage := 'Syntax error during interpretation';
	END_IF
	IF NC_Error_Code = 16#4113 THEN
		stErrorMessage := 'Missing subroutine';
	END_IF
	IF NC_Error_Code = 16#4114 THEN
		stErrorMessage := 'Loading buffer of interpreter is too small';
	END_IF
	IF NC_Error_Code = 16#4115 THEN
		stErrorMessage := 'Symbolic“  - reserved';
	END_IF
	IF NC_Error_Code = 16#4116 THEN
		stErrorMessage := 'Symbolic“  - reserved';
	END_IF
	IF NC_Error_Code = 16#4117 THEN
		stErrorMessage := 'Subroutine incomplete';
	END_IF
	IF NC_Error_Code = 16#4120 THEN
		stErrorMessage := 'Divide by zero';
	END_IF
	IF NC_Error_Code = 16#4121 THEN
		stErrorMessage := 'Invalid circle parameterisation';
	END_IF
	IF NC_Error_Code = 16#4122 THEN
		stErrorMessage := 'Invalid FPU-Operation';
	END_IF
	IF NC_Error_Code = 16#4130 THEN
		stErrorMessage := 'Stack overflow: subroutines';
	END_IF
	IF NC_Error_Code = 16#4131 THEN
		stErrorMessage := 'Stack underflow: subroutines';
	END_IF
	IF NC_Error_Code = 16#4132 THEN
		stErrorMessage := 'Stack overflow: arithmetic unit';
	END_IF
	IF NC_Error_Code = 16#4133 THEN
		stErrorMessage := 'Stack underflow: arithmetic unit';
	END_IF
	IF NC_Error_Code = 16#4140 THEN
		stErrorMessage := 'Register index not allowed';
	END_IF
	IF NC_Error_Code = 16#4141 THEN
		stErrorMessage := 'Unacceptable G-function index';
	END_IF
	IF NC_Error_Code = 16#4142 THEN
		stErrorMessage := 'Unacceptable M-function index';
	END_IF
	IF NC_Error_Code = 16#4143 THEN
		stErrorMessage := 'Unacceptable extended address';
	END_IF
	IF NC_Error_Code = 16#4144 THEN
		stErrorMessage := 'Unacceptable index to the internal H-function';
	END_IF
	IF NC_Error_Code = 16#4145 THEN
		stErrorMessage := 'Machine data value unacceptable';
	END_IF
	IF NC_Error_Code = 16#4150 THEN
		stErrorMessage := 'Cannot change tool params here';
	END_IF
	IF NC_Error_Code = 16#4151 THEN
		stErrorMessage := 'Cannot calculate tool compensation';
	END_IF
	IF NC_Error_Code = 16#4152 THEN
		stErrorMessage := 'Tool compensation: The plane for the tool compensation cannot be changed here.';
	END_IF
	IF NC_Error_Code = 16#4153 THEN
		stErrorMessage := 'Tool compensation:  The D-Word is missing or invalid by turning on the tool compensation. ';
	END_IF
	IF NC_Error_Code = 16#4154 THEN
		stErrorMessage := 'Tool compensation:  The spezified tool radius is invalid because the value is less or equal zero.';
	END_IF
	IF NC_Error_Code = 16#4155 THEN
		stErrorMessage := 'Tool compensation: The tool radius cannot be changed here ';
	END_IF
	IF NC_Error_Code = 16#4156 THEN
		stErrorMessage := 'Tool compensation:  Collision Detection Table is full.';
	END_IF
	IF NC_Error_Code = 16#4157 THEN
		stErrorMessage := 'Tool compensation: Internal error while turning on the contour collision detection. ';
	END_IF
	IF NC_Error_Code = 16#4158 THEN
		stErrorMessage := 'Tool compensation:  Internal error within the contour collision detection - update reversed geo failed.';
	END_IF
	IF NC_Error_Code = 16#4159 THEN
		stErrorMessage := 'Tool compensation:  Unexpected combination of geometrie types by active contour collision detection.';
	END_IF
	IF NC_Error_Code = 16#415A THEN
		stErrorMessage := 'Tool compensation: Programmed inner circle is smaller than the cutter radius';
	END_IF
	IF NC_Error_Code = 16#415B THEN
		stErrorMessage := 'Tool compensation:  Bottle neck detection recognized contour violation';
	END_IF
	IF NC_Error_Code = 16#415C THEN
		stErrorMessage := 'Table for corrected entries is full';
	END_IF
	IF NC_Error_Code = 16#415D THEN
		stErrorMessage := 'Input table for tangential following is full';
	END_IF
	IF NC_Error_Code = 16#415E THEN
		stErrorMessage := 'Executing table for tangential following is full';
	END_IF
	IF NC_Error_Code = 16#415F THEN
		stErrorMessage := 'Geometric entry for tangential following can not be calculated';
	END_IF
	IF NC_Error_Code = 16#4160 THEN
		stErrorMessage := 'reserved';
	END_IF
	IF NC_Error_Code = 16#4161 THEN
		stErrorMessage := 'reserved';
	END_IF
	IF NC_Error_Code = 16#4162 THEN
		stErrorMessage := 'The acutal active interpolation rules (g-code), zero-shifts, or rotation cannot be detected';
	END_IF
END_IF

(*Group Errors*)
IF dwMask = 16#42 THEN
	stGroupMessage := 'Group Error: ';
	IF NC_Error_Code = 16#4200 THEN
		stErrorMessage := 'Group ID not allowed';
	END_IF
	IF NC_Error_Code = 16#4201 THEN
		stErrorMessage := 'Group type not allowed';
	END_IF
	IF NC_Error_Code = 16#4202 THEN
		stErrorMessage := 'Master axis index not allowed';
	END_IF
	IF NC_Error_Code = 16#4203 THEN
		stErrorMessage := 'Slave axis index not allowed';
	END_IF
	IF NC_Error_Code = 16#4204 THEN
		stErrorMessage := 'GROUPERR_INTERNAL ';
	END_IF
	IF NC_Error_Code = 16#4205 THEN
		stErrorMessage := 'Invalid cycle time for statement execution task (SAF)';
	END_IF
	IF NC_Error_Code = 16#4206 THEN
		stErrorMessage := 'GROUPERR_RANGE_MAXELEMENTSINAXIS ';
	END_IF
	IF NC_Error_Code = 16#4207 THEN
		stErrorMessage := 'Invalid cycle time for the statement preparation task (SVB)';
	END_IF
	IF NC_Error_Code = 16#4208 THEN
		stErrorMessage := 'Single step mode not allowed';
	END_IF
	IF NC_Error_Code = 16#4209 THEN
		stErrorMessage := 'Group deactivation not allowed';
	END_IF
	IF NC_Error_Code = 16#420A THEN
		stErrorMessage := 'Statement execution state (SAF state) not allowed';
	END_IF
	IF NC_Error_Code = 16#420B THEN
		stErrorMessage := 'Chanel address';
	END_IF
	IF NC_Error_Code = 16#420C THEN
		stErrorMessage := 'Axis address (master axis)';
	END_IF
	IF NC_Error_Code = 16#420D THEN
		stErrorMessage := 'Master axis address';
	END_IF
	IF NC_Error_Code = 16#420E THEN
		stErrorMessage := 'Slave axis address';
	END_IF
	IF NC_Error_Code = 16#420F THEN
		stErrorMessage := 'Slave set value generator address';
	END_IF
	IF NC_Error_Code = 16#4210 THEN
		stErrorMessage := 'Encoder address';
	END_IF
	IF NC_Error_Code = 16#4211 THEN
		stErrorMessage := 'Controller address';
	END_IF
	IF NC_Error_Code = 16#4212 THEN
		stErrorMessage := 'Drive address';
	END_IF
	IF NC_Error_Code = 16#4213 THEN
		stErrorMessage := 'GROUPERR_ADDR_MASTERGENERATOR';
	END_IF
	IF NC_Error_Code = 16#4214 THEN
		stErrorMessage := 'Axis interface NC to PLC address';
	END_IF
	IF NC_Error_Code = 16#4215 THEN
		stErrorMessage := 'Slave axis address';
	END_IF
	IF NC_Error_Code = 16#4216 THEN
		stErrorMessage := 'Table adress unknown';
	END_IF
	IF NC_Error_Code = 16#4217 THEN
		stErrorMessage := 'NcControl address';
	END_IF
	IF NC_Error_Code = 16#4218 THEN
		stErrorMessage := 'Axis is blocked for commands while persistent NC data are queued';
	END_IF
	IF NC_Error_Code = 16#421A THEN
		stErrorMessage := 'The master axis start position does not permit synchronisation';
	END_IF
	IF NC_Error_Code = 16#421B THEN
		stErrorMessage := 'Slave coupling factor (gearing factor) of 0.0 is not allowed';
	END_IF
	IF NC_Error_Code = 16#421C THEN
		stErrorMessage := 'Insertion of master axis into group not allowed';
	END_IF
	IF NC_Error_Code = 16#421D THEN
		stErrorMessage := 'Deletion of master axis from group not allowed';
	END_IF
	IF NC_Error_Code = 16#421E THEN
		stErrorMessage := 'Function/feature is not supported from the setpoint generator ';
	END_IF
	IF NC_Error_Code = 16#421F THEN
		stErrorMessage := 'Group initialisation';
	END_IF
	IF NC_Error_Code = 16#4220 THEN
		stErrorMessage := 'Group not ready / group not ready for new task';
	END_IF
	IF NC_Error_Code = 16#4221 THEN
		stErrorMessage := 'Requested set velocity is not allowed';
	END_IF
	IF NC_Error_Code = 16#4222 THEN
		stErrorMessage := 'Requested target position is not allowed (master axis)';
	END_IF
	IF NC_Error_Code = 16#4223 THEN
		stErrorMessage := 'No enable for controller and/or feed (Master axis)';
	END_IF
	IF NC_Error_Code = 16#4224 THEN
		stErrorMessage := 'Movement smaller than one encoder increment';
	END_IF
	IF NC_Error_Code = 16#4225 THEN
		stErrorMessage := 'Drive not ready during axis start';
	END_IF
	IF NC_Error_Code = 16#4226 THEN
		stErrorMessage := 'Invalid parameters of the emergency stop.';
	END_IF
	IF NC_Error_Code = 16#4227 THEN
		stErrorMessage := 'The setpoint generator is inactive such that no instructions are accepted';
	END_IF
	IF NC_Error_Code = 16#4228 THEN
		stErrorMessage := 'Requested traverse distance is not allowed';
	END_IF
	IF NC_Error_Code = 16#4229 THEN
		stErrorMessage := 'Requested target position is not allowed (slave axis)';
	END_IF
	IF NC_Error_Code = 16#422A THEN
		stErrorMessage := 'No enable for controller and/or feed (slave axis)';
	END_IF
	IF NC_Error_Code = 16#422B THEN
		stErrorMessage := 'The activation position (position threshold) is out of range of the actual positioning';
	END_IF
	IF NC_Error_Code = 16#422C THEN
		stErrorMessage := 'The start or activation data of the external setpoint generation are not valid';
	END_IF
	IF NC_Error_Code = 16#422D THEN
		stErrorMessage := 'Velocity is not constant';
	END_IF
	IF NC_Error_Code = 16#422E THEN
		stErrorMessage := 'Jerk less than or equal to 0.0 is not allowed';
	END_IF
	IF NC_Error_Code = 16#422F THEN
		stErrorMessage := 'Acceleration less than or equal to 0.0 is not allowed';
	END_IF
	IF NC_Error_Code = 16#4230 THEN
		stErrorMessage := 'Absolute deceleration value less than or equal to 0.0 is not allowed';
	END_IF
	IF NC_Error_Code = 16#4231 THEN
		stErrorMessage := 'Set velocity less than or equal to 0.0 is not allowed';
	END_IF
	IF NC_Error_Code = 16#4232 THEN
		stErrorMessage := 'Loss of precision when trying a positioning';
	END_IF
	IF NC_Error_Code = 16#4233 THEN
		stErrorMessage := 'Cycle time less than or equal to 0.0 is not allowed';
	END_IF
	IF NC_Error_Code = 16#4234 THEN
		stErrorMessage := 'PTP data type <intasdouble> range exceeded';
	END_IF
	IF NC_Error_Code = 16#4235 THEN
		stErrorMessage := 'PTP LHL velocity profile cannot be generated';
	END_IF
	IF NC_Error_Code = 16#4236 THEN
		stErrorMessage := 'PTP HML velocity profile cannot be generated';
	END_IF
	IF NC_Error_Code = 16#4237 THEN
		stErrorMessage := 'Start data address is invalid';
	END_IF
	IF NC_Error_Code = 16#4238 THEN
		stErrorMessage := 'Velocity override (start override) is not allowed';
	END_IF
	IF NC_Error_Code = 16#4239 THEN
		stErrorMessage := 'Start type not allowed';
	END_IF
	IF NC_Error_Code = 16#423A THEN
		stErrorMessage := 'Velocity overflow (overshoot in the velocity)';
	END_IF
	IF NC_Error_Code = 16#423B THEN
		stErrorMessage := 'Start parameter for the axis structure is invalid';
	END_IF
	IF NC_Error_Code = 16#423C THEN
		stErrorMessage := 'Override generator initialisation parameter invalid';
	END_IF
	IF NC_Error_Code = 16#423D THEN
		stErrorMessage := 'Slave axis has not set value generator';
	END_IF
	IF NC_Error_Code = 16#423E THEN
		stErrorMessage := 'Table is empty';
	END_IF
	IF NC_Error_Code = 16#423F THEN
		stErrorMessage := 'Table is full';
	END_IF
	IF NC_Error_Code = 16#4240 THEN
		stErrorMessage := 'No memory available';
	END_IF
	IF NC_Error_Code = 16#4241 THEN
		stErrorMessage := 'Table already contains an entry';
	END_IF
	IF NC_Error_Code = 16#4242 THEN
		stErrorMessage := 'Stop is already active';
	END_IF
	IF NC_Error_Code = 16#4243 THEN
		stErrorMessage := 'Compensation has not been carried out over the full compensation section';
	END_IF
	IF NC_Error_Code = 16#4244 THEN
		stErrorMessage := 'Start parameter address for the compensation invalid';
	END_IF
	IF NC_Error_Code = 16#4245 THEN
		stErrorMessage := 'Compensation active';
	END_IF
	IF NC_Error_Code = 16#4246 THEN
		stErrorMessage := 'Compensation not active';
	END_IF
	IF NC_Error_Code = 16#4247 THEN
		stErrorMessage := 'Compensation type invalid';
	END_IF
	IF NC_Error_Code = 16#4248 THEN
		stErrorMessage := 'Axis address for compensation invalid';
	END_IF
	IF NC_Error_Code = 16#4249 THEN
		stErrorMessage := 'Invalid slave address';
	END_IF
	IF NC_Error_Code = 16#424A THEN
		stErrorMessage := 'Coupling velocity invalid';
	END_IF
	IF NC_Error_Code = 16#424B THEN
		stErrorMessage := 'Coupling velocities not constant';
	END_IF
	IF NC_Error_Code = 16#424C THEN
		stErrorMessage := 'Cycle time less than or equal to 0.0 is not allowed';
	END_IF
	IF NC_Error_Code = 16#424D THEN
		stErrorMessage := 'Decoupling task not allowed';
	END_IF
	IF NC_Error_Code = 16#424E THEN
		stErrorMessage := 'Function not allowed';
	END_IF
	IF NC_Error_Code = 16#424F THEN
		stErrorMessage := 'No valid table weighting has been set';
	END_IF
	IF NC_Error_Code = 16#4250 THEN
		stErrorMessage := 'Axis type, actual position type or end position type is not allowed';
	END_IF
	IF NC_Error_Code = 16#4251 THEN
		stErrorMessage := 'Function not presently supported';
	END_IF
	IF NC_Error_Code = 16#4252 THEN
		stErrorMessage := 'State of state machine invalid';
	END_IF
	IF NC_Error_Code = 16#4253 THEN
		stErrorMessage := 'Reference cam became free too soon';
	END_IF
	IF NC_Error_Code = 16#4254 THEN
		stErrorMessage := 'Clearance monitoring between activation of the hardware latch and appearance of the sync pulse';
	END_IF
	IF NC_Error_Code = 16#4255 THEN
		stErrorMessage := 'No memory available';
	END_IF
	IF NC_Error_Code = 16#4256 THEN
		stErrorMessage := 'The table slave axis has no active table';
	END_IF
	IF NC_Error_Code = 16#4257 THEN
		stErrorMessage := 'Function not allowed';
	END_IF
	IF NC_Error_Code = 16#4258 THEN
		stErrorMessage := 'Stopping compensation not allowed';
	END_IF
	IF NC_Error_Code = 16#4259 THEN
		stErrorMessage := 'Slave table is being used';
	END_IF
	IF NC_Error_Code = 16#425A THEN
		stErrorMessage := 'Master or slave axis is processing a job (e.g. positioning command) while coupling is requested';
	END_IF
	IF NC_Error_Code = 16#425B THEN
		stErrorMessage := 'Slave (start) parameter is incorrect';
	END_IF
	IF NC_Error_Code = 16#425C THEN
		stErrorMessage := 'Slave type is incorrect';
	END_IF
	IF NC_Error_Code = 16#425D THEN
		stErrorMessage := 'Axis stop is already active';
	END_IF
	IF NC_Error_Code = 16#425E THEN
		stErrorMessage := 'Compensation refused';
	END_IF
	IF NC_Error_Code = 16#425F THEN
		stErrorMessage := 'Compensation not started';
	END_IF
	IF NC_Error_Code = 16#4260 THEN
		stErrorMessage := 'Controller enable';
	END_IF
	IF NC_Error_Code = 16#4261 THEN
		stErrorMessage := 'Table not found';
	END_IF
	IF NC_Error_Code = 16#4262 THEN
		stErrorMessage := 'Incorrect table type';
	END_IF
	IF NC_Error_Code = 16#4263 THEN
		stErrorMessage := 'Single step mode';
	END_IF
	IF NC_Error_Code = 16#4264 THEN
		stErrorMessage := 'Group task unknown (asynchronous table entry)';
	END_IF
	IF NC_Error_Code = 16#4265 THEN
		stErrorMessage := 'Group function unknown (synchronous function)';
	END_IF
	IF NC_Error_Code = 16#4266 THEN
		stErrorMessage := 'Group task for slave not allowed';
	END_IF
	IF NC_Error_Code = 16#4267 THEN
		stErrorMessage := 'Group function for slave not allowed';
	END_IF
	IF NC_Error_Code = 16#4268 THEN
		stErrorMessage := 'GROUPERR_GROUPFUNC_NOMOTION';
	END_IF
	IF NC_Error_Code = 16#4269 THEN
		stErrorMessage := 'Startposition=Setpoint Position';
	END_IF
	IF NC_Error_Code = 16#426A THEN
		stErrorMessage := 'Parameters of the delay-denerator are invalid';
	END_IF
	IF NC_Error_Code = 16#426B THEN
		stErrorMessage := 'External parameters of the superimposed instruction are invalid';
	END_IF
	IF NC_Error_Code = 16#426C THEN
		stErrorMessage := 'Invalid overridetype';
	END_IF
	IF NC_Error_Code = 16#426D THEN
		stErrorMessage := 'Activation position under/overrun';
	END_IF
	IF NC_Error_Code = 16#426E THEN
		stErrorMessage := 'Activation impossible: Master is standing';
	END_IF
	IF NC_Error_Code = 16#426F THEN
		stErrorMessage := 'Activation mode not possible';
	END_IF
	IF NC_Error_Code = 16#4270 THEN
		stErrorMessage := 'Start parameter for the compensation is invalid';
	END_IF
	IF NC_Error_Code = 16#4271 THEN
		stErrorMessage := 'Start parameter for the compensation is invalid';
	END_IF
	IF NC_Error_Code = 16#4272 THEN
		stErrorMessage := 'Start parameter for the compensation is invalid';
	END_IF
	IF NC_Error_Code = 16#4273 THEN
		stErrorMessage := 'Target position under/overrun';
	END_IF
	IF NC_Error_Code = 16#4274 THEN
		stErrorMessage := 'Target position will be under/overrun';
	END_IF
	IF NC_Error_Code = 16#4276 THEN
		stErrorMessage := 'GROUPERR_GUIDERSTARTDATA';
	END_IF
	IF NC_Error_Code = 16#4279 THEN
		stErrorMessage := 'GROUPERR_GUIDEROVERRUN';
	END_IF
	IF NC_Error_Code = 16#427A THEN
		stErrorMessage := 'GROUPERR_GUIDERLOOKAHEAD';
	END_IF
	IF NC_Error_Code = 16#427B THEN
		stErrorMessage := 'GROUPERR_GUIDERLOOKAHEADEND';
	END_IF
	IF NC_Error_Code = 16#427C THEN
		stErrorMessage := 'GROUPERR_GUIDERLOOKAHEADREQU';
	END_IF
	IF NC_Error_Code = 16#427D THEN
		stErrorMessage := 'GROUPERR_GUIDERMODE';
	END_IF
	IF NC_Error_Code = 16#427E THEN
		stErrorMessage := 'A requested motion command could not be realized (BISECTION)';
	END_IF
	IF NC_Error_Code = 16#427F THEN
		stErrorMessage := 'The new target position either has been overrun or will be overrun';
	END_IF
	IF NC_Error_Code = 16#4280 THEN
		stErrorMessage := 'Group not ready / group not ready for new task';
	END_IF
	IF NC_Error_Code = 16#4281 THEN
		stErrorMessage := 'The parameters of the oriented stop (O-Stop) are not admitted.';
	END_IF
	IF NC_Error_Code = 16#4282 THEN
		stErrorMessage := 'The modulo target position of the modulo-start is invalid';
	END_IF
	IF NC_Error_Code = 16#4283 THEN
		stErrorMessage := 'The online change activation mode is invalid';
	END_IF
	IF NC_Error_Code = 16#4284 THEN
		stErrorMessage := 'The parameterized jerk rate is not permitted';
	END_IF
	IF NC_Error_Code = 16#4285 THEN
		stErrorMessage := 'The parameterized acceleration or deceleration is not permitted';
	END_IF
	IF NC_Error_Code = 16#4286 THEN
		stErrorMessage := 'The parameterized velocity is not permitted';
	END_IF
	IF NC_Error_Code = 16#4287 THEN
		stErrorMessage := 'A activation cannot be executed due to a pending activation';
	END_IF
	IF NC_Error_Code = 16#4288 THEN
		stErrorMessage := 'Illegal combination of different cycle times within an axis group';
	END_IF
	IF NC_Error_Code = 16#4289 THEN
		stErrorMessage := 'Illegal motion reversal';
	END_IF
	IF NC_Error_Code = 16#428A THEN
		stErrorMessage := 'Illegal moment for an axis command because there is an old axis command with activation position still active';
	END_IF
	IF NC_Error_Code = 16#428B THEN
		stErrorMessage := 'Error in the stop-calculation routine';
	END_IF
	IF NC_Error_Code = 16#428C THEN
		stErrorMessage := 'A command with activation position cannot fully be performed because the remaining path is too short';
	END_IF
	IF NC_Error_Code = 16#428D THEN
		stErrorMessage := 'Illegal decoupletype when decoupling a slave axis';
	END_IF
	IF NC_Error_Code = 16#428E THEN
		stErrorMessage := 'Illegal target velocity when decoupling a slave axis';
	END_IF
	IF NC_Error_Code = 16#428F THEN
		stErrorMessage := 'The command new dynamic parameter cannot be performed since this would require a new target velocity';
	END_IF
	IF NC_Error_Code = 16#4290 THEN
		stErrorMessage := 'A command with activation position cannot be performed becaus the axis is already in the brake phase';
	END_IF
	IF NC_Error_Code = 16#4291 THEN
		stErrorMessage := 'Decouple routine of slave axis does not return a valid solution';
	END_IF
	IF NC_Error_Code = 16#4292 THEN
		stErrorMessage := 'Command not be executed because the command buffer is full filled';
	END_IF
	IF NC_Error_Code = 16#4293 THEN
		stErrorMessage := 'Command is rejected due to an internal error in the Look Ahead';
	END_IF
	IF NC_Error_Code = 16#4294 THEN
		stErrorMessage := 'Command is rejected because the segment target velocity is not realized';
	END_IF
	IF NC_Error_Code = 16#4295 THEN
		stErrorMessage := 'Command is rejected because the segment start velocity or the segment end velocity is not allowed';
	END_IF
	IF NC_Error_Code = 16#4296 THEN
		stErrorMessage := 'Logical positioning direction is inconsistent with the direction of the buffer command';
	END_IF
	IF NC_Error_Code = 16#4297 THEN
		stErrorMessage := 'Command is rejected because the remaining positioning length is to small';
	END_IF
	IF NC_Error_Code = 16#42A0 THEN
		stErrorMessage := 'Group/axis consequential error';
	END_IF
	IF NC_Error_Code = 16#42A1 THEN
		stErrorMessage := 'Velocity reduction factor for C0/C1 transition is not allowed';
	END_IF
	IF NC_Error_Code = 16#42A2 THEN
		stErrorMessage := 'Critical angle at segment transition not allowed';
	END_IF
	IF NC_Error_Code = 16#42A3 THEN
		stErrorMessage := 'Radius of the tolerance sphere" (NOT IMPLEMENTED)   ';
	END_IF
	IF NC_Error_Code = 16#42A5 THEN
		stErrorMessage := 'Start type';
	END_IF
	IF NC_Error_Code = 16#42A9 THEN
		stErrorMessage := 'Curve velocity reduction method not allowed';
	END_IF
	IF NC_Error_Code = 16#42AA THEN
		stErrorMessage := 'Minimum velocity not allowed';
	END_IF
	IF NC_Error_Code = 16#42AB THEN
		stErrorMessage := 'Power function input not allowed';
	END_IF
	IF NC_Error_Code = 16#42AC THEN
		stErrorMessage := 'Dynamic change parameter not allowed';
	END_IF
	IF NC_Error_Code = 16#42AD THEN
		stErrorMessage := 'Memory allocation error';
	END_IF
	IF NC_Error_Code = 16#4AE THEN
		stErrorMessage := 'The calculated end position differs from the end position in the nc instruction ';
	END_IF
	IF NC_Error_Code = 16#42AF THEN
		stErrorMessage := 'Calculate remaining chord length';
	END_IF
	IF NC_Error_Code = 16#42B0 THEN
		stErrorMessage := 'Set value generator SVB active';
	END_IF
	IF NC_Error_Code = 16#42B1 THEN
		stErrorMessage := 'SVB parameter not allowed';
	END_IF
	IF NC_Error_Code = 16#42B2 THEN
		stErrorMessage := 'Velocity reduction factor not allowed';
	END_IF
	IF NC_Error_Code = 16#42B3 THEN
		stErrorMessage := 'Helix is a circle';
	END_IF
	IF NC_Error_Code = 16#42B4 THEN
		stErrorMessage := 'Helix is a straight line';
	END_IF
	IF NC_Error_Code = 16#42B5 THEN
		stErrorMessage := 'Guider parameter not allowed';
	END_IF
	IF NC_Error_Code = 16#42B6 THEN
		stErrorMessage := 'Invalid segment address';
	END_IF
	IF NC_Error_Code = 16#42B7 THEN
		stErrorMessage := 'Unparametrised generator';
	END_IF
	IF NC_Error_Code = 16#42B8 THEN
		stErrorMessage := 'Unparametrised table';
	END_IF
	IF NC_Error_Code = 16#42BA THEN
		stErrorMessage := 'The calculation of the arc length of the smoothed path failed ';
	END_IF
	IF NC_Error_Code = 16#42BB THEN
		stErrorMessage := 'The radius of the tolerance ball is too small (smaller than 0.1 mm).';
	END_IF
	IF NC_Error_Code = 16#42BD THEN
		stErrorMessage := 'NC-Block violates software limit switches of the group';
	END_IF
	IF NC_Error_Code = 16#42BE THEN
		stErrorMessage := 'GROUPERR_DXD_SOFTENDCHECK';
	END_IF
	IF NC_Error_Code = 16#42BF THEN
		stErrorMessage := 'GROUPERR_DXD_RTTG_VELOREFERENCE';
	END_IF
	IF NC_Error_Code = 16#42C0 THEN
		stErrorMessage := 'Interpolating group contains axes of an incorrect axis type';
	END_IF
	IF NC_Error_Code = 16#42C1 THEN
		stErrorMessage := 'Scalar product can not be calculated';
	END_IF
	IF NC_Error_Code = 16#42C2 THEN
		stErrorMessage := 'Inverse cosine can not be calculated';
	END_IF
	IF NC_Error_Code = 16#42C3 THEN
		stErrorMessage := 'Invalid table entry type';
	END_IF
	IF NC_Error_Code = 16#42C4 THEN
		stErrorMessage := 'Invalid DIN66025 information type';
	END_IF
	IF NC_Error_Code = 16#42C5 THEN
		stErrorMessage := 'Invalid dimension';
	END_IF
	IF NC_Error_Code = 16#42C6 THEN
		stErrorMessage := 'Geometrical object is not a straight line';
	END_IF
	IF NC_Error_Code = 16#42C7 THEN
		stErrorMessage := 'Geometrical object is not a circle';
	END_IF
	IF NC_Error_Code = 16#42C8 THEN
		stErrorMessage := 'Geometrical object is not a helix';
	END_IF
	IF NC_Error_Code = 16#42C9 THEN
		stErrorMessage := 'Set velocity less than or equal to 0.0 is invalid';
	END_IF
	IF NC_Error_Code = 16#42CA THEN
		stErrorMessage := 'Address for look-ahead invalid';
	END_IF
	IF NC_Error_Code = 16#42CB THEN
		stErrorMessage := 'Set value generator SAF active';
	END_IF
	IF NC_Error_Code = 16#42CC THEN
		stErrorMessage := 'CNC set value generation not active';
	END_IF
	IF NC_Error_Code = 16#42CD THEN
		stErrorMessage := 'CNC set value generation in the stop phase';
	END_IF
	IF NC_Error_Code = 16#42CE THEN
		stErrorMessage := 'Override not allowed';
	END_IF
	IF NC_Error_Code = 16#42CF THEN
		stErrorMessage := 'Invalid table address';
	END_IF
	IF NC_Error_Code = 16#42D0 THEN
		stErrorMessage := 'Invalid table entry type';
	END_IF
	IF NC_Error_Code = 16#42D1 THEN
		stErrorMessage := 'Memory allocation failed" Memory allocation for the table has failed. ';
	END_IF
	IF NC_Error_Code = 16#42D2 THEN
		stErrorMessage := 'Memory allocation failed" Memory allocation for the filter has failed. ';
	END_IF
	IF NC_Error_Code = 16#42D3 THEN
		stErrorMessage := 'Invalid parameter" Filter parameter is not allowed. ';
	END_IF
	IF NC_Error_Code = 16#42D4 THEN
		stErrorMessage := 'Delete Distance To Go failed';
	END_IF
	IF NC_Error_Code = 16#42D5 THEN
		stErrorMessage := 'The setpoint generator of the fying saw generates incompatible values';
	END_IF
	IF NC_Error_Code = 16#42D6 THEN
		stErrorMessage := 'Axis will be stopped since otherwise it will overrun its target position (old PTP setpoint generator)';
	END_IF
	IF NC_Error_Code = 16#42D7 THEN
		stErrorMessage := 'Internal error in the transformation from slave to master';
	END_IF
	IF NC_Error_Code = 16#42D8 THEN
		stErrorMessage := 'Wrong direction in the transformation of slave to master';
	END_IF
	IF NC_Error_Code = 16#42DA THEN
		stErrorMessage := 'Parameter of Motion Function (MF) table incorrect';
	END_IF
	IF NC_Error_Code = 16#42DB THEN
		stErrorMessage := 'Parameter of Motion Function (MF) table invalid';
	END_IF
	IF NC_Error_Code = 16#42DC THEN
		stErrorMessage := 'Internal error by using Motion Function (MF)';
	END_IF
	IF NC_Error_Code = 16#42DD THEN
		stErrorMessage := 'Axis coupling with synchronization generator declined because of incorrect axis dynamic values';
	END_IF
	IF NC_Error_Code = 16#42DE THEN
		stErrorMessage := 'Coupling conditions of synchronization generator incorrect';
	END_IF
	IF NC_Error_Code = 16#42DF THEN
		stErrorMessage := 'Moving profile of synchronization generator declines dynamic limit of slave axis or required characterstic of profile';
	END_IF
	IF NC_Error_Code = 16#42E0 THEN
		stErrorMessage := 'Invalid parameter" The encoder generator parameter is not allowed. ';
	END_IF
	IF NC_Error_Code = 16#42E1 THEN
		stErrorMessage := 'Invalid parameter" The external (Fifo) generator parameter is not allowed. ';
	END_IF
	IF NC_Error_Code = 16#42E2 THEN
		stErrorMessage := 'External generator is active';
	END_IF
	IF NC_Error_Code = 16#42E3 THEN
		stErrorMessage := 'External generator is not active';
	END_IF
	IF NC_Error_Code = 16#42E4 THEN
		stErrorMessage := 'NC-Block with auxiliary axis violates software limit switches of the group';
	END_IF
	IF NC_Error_Code = 16#42E5 THEN
		stErrorMessage := 'NC-Block type Bezier spline curve contains a cusp (singularity)';
	END_IF
	IF NC_Error_Code = 16#42E7 THEN
		stErrorMessage := 'Value for dead time compensation not allowed';
	END_IF
	IF NC_Error_Code = 16#42E8 THEN
		stErrorMessage := 'GROUPERR_RANGE_NOMOTIONWINDOW';
	END_IF
	IF NC_Error_Code = 16#42E9 THEN
		stErrorMessage := 'GROUPERR_RANGE_NOMOTIONFILTERTIME';
	END_IF
	IF NC_Error_Code = 16#42EA THEN
		stErrorMessage := 'GROUPERR_RANGE_TIMEUNITFIFO';
	END_IF
	IF NC_Error_Code = 16#42EB THEN
		stErrorMessage := 'GROUPERR_RANGE_OVERRIDETYPE';
	END_IF
	IF NC_Error_Code = 16#42EC THEN
		stErrorMessage := 'GROUPERR_RANGE_OVERRIDECHANGETIME';
	END_IF
	IF NC_Error_Code = 16#42ED THEN
		stErrorMessage := 'GROUPERR_FIFO_INVALIDDIMENSION';
	END_IF
	IF NC_Error_Code = 16#42EE THEN
		stErrorMessage := 'GROUPERR_ADDR_FIFOTABLE';
	END_IF
	IF NC_Error_Code = 16#42EF THEN
		stErrorMessage := 'Axis is locked for motion commands because a stop command is still active';
	END_IF
	IF NC_Error_Code = 16#42F0 THEN
		stErrorMessage := 'Invalid number of auxiliary axes';
	END_IF
	IF NC_Error_Code = 16#42F1 THEN
		stErrorMessage := 'Invalid reduction parameter for auxiliary axes';
	END_IF
	IF NC_Error_Code = 16#42F2 THEN
		stErrorMessage := 'Invalid dynamic parameter for auxiliary axes';
	END_IF
	IF NC_Error_Code = 16#42F3 THEN
		stErrorMessage := 'Invalid coupling parameter for auxiliary axes';
	END_IF
	IF NC_Error_Code = 16#42F4 THEN
		stErrorMessage := 'Invalid auxiliary axis entry';
	END_IF
	IF NC_Error_Code = 16#42FF THEN
		stErrorMessage := 'GROUPERR_HYMMEN_WATCHDOG';
	END_IF
END_IF

(*Axis Errors*)
IF dwMask = 16#43 THEN
	stGroupMessage := 'Axis Error: ';
	IF NC_Error_Code = 16#4300 THEN
		stErrorMessage := 'Axis ID not allowed';
	END_IF
	IF NC_Error_Code = 16#4301 THEN
		stErrorMessage := 'Axis type not allowed';
	END_IF
	IF NC_Error_Code = 16#4306 THEN
		stErrorMessage := 'Slow manual velocity not allowed';
	END_IF
	IF NC_Error_Code = 16#4307 THEN
		stErrorMessage := 'Fast manual velocity NOT allowed';
	END_IF
	IF NC_Error_Code = 16#4308 THEN
		stErrorMessage := 'High speed not allowed';
	END_IF
	IF NC_Error_Code = 16#4309 THEN
		stErrorMessage := 'Acceleration not allowed';
	END_IF
	IF NC_Error_Code = 16#430A THEN
		stErrorMessage := 'Deceleration not allowed';
	END_IF
	IF NC_Error_Code = 16#430B THEN
		stErrorMessage := 'Jerk not allowed';
	END_IF
	IF NC_Error_Code = 16#430C THEN
		stErrorMessage := 'Delay time between position and velocity is not allowed';
	END_IF
	IF NC_Error_Code = 16#430D THEN
		stErrorMessage := 'Override-Type not allowed';
	END_IF
	IF NC_Error_Code = 16#4312 THEN
		stErrorMessage := 'Referencing velocity in direction of cam not allowed';
	END_IF
	IF NC_Error_Code = 16#4313 THEN
		stErrorMessage := 'Referencing velocity in sync direction not allowed';
	END_IF
	IF NC_Error_Code = 16#4314 THEN
		stErrorMessage := 'Pulse width in positive direction not allowed';
	END_IF
	IF NC_Error_Code = 16#4315 THEN
		stErrorMessage := 'Pulse width in negative direction not allowed';
	END_IF
	IF NC_Error_Code = 16#4316 THEN
		stErrorMessage := 'Pulse time in positive direction not allowed';
	END_IF
	IF NC_Error_Code = 16#4317 THEN
		stErrorMessage := 'Pulse time in negative direction not allowed';
	END_IF
	IF NC_Error_Code = 16#4318 THEN
		stErrorMessage := 'Creep distance in positive direction not allowed';
	END_IF
	IF NC_Error_Code = 16#4319 THEN
		stErrorMessage := 'Creep distance in negative direction not allowed';
	END_IF
	IF NC_Error_Code = 16#431A THEN
		stErrorMessage := 'Braking distance in positive direction not allowed';
	END_IF
	IF NC_Error_Code = 16#431B THEN
		stErrorMessage := 'Braking distance in negative direction not allowed';
	END_IF
	IF NC_Error_Code = 16#431C THEN
		stErrorMessage := 'Braking time in positive direction not allowed';
	END_IF
	IF NC_Error_Code = 16#431D THEN
		stErrorMessage := 'Braking time in negative direction not allowed';
	END_IF
	IF NC_Error_Code = 16#431E THEN
		stErrorMessage := 'Switching time from high to low speed not allowed';
	END_IF
	IF NC_Error_Code = 16#431F THEN
		stErrorMessage := 'Creep distance for stop not allowed';
	END_IF
	IF NC_Error_Code = 16#4320 THEN
		stErrorMessage := 'Motion monitoring not allowed';
	END_IF
	IF NC_Error_Code = 16#4321 THEN
		stErrorMessage := 'Position window monitoring not allowed';
	END_IF
	IF NC_Error_Code = 16#4322 THEN
		stErrorMessage := 'Target window monitoring not allowed';
	END_IF
	IF NC_Error_Code = 16#4323 THEN
		stErrorMessage := 'Loop not allowed';
	END_IF
	IF NC_Error_Code = 16#4324 THEN
		stErrorMessage := 'Motion monitoring time not allowed';
	END_IF
	IF NC_Error_Code = 16#4325 THEN
		stErrorMessage := 'Target window range not allowed';
	END_IF
	IF NC_Error_Code = 16#4326 THEN
		stErrorMessage := 'Position window range not allowed';
	END_IF
	IF NC_Error_Code = 16#4327 THEN
		stErrorMessage := 'Position window monitoring time not allowed';
	END_IF
	IF NC_Error_Code = 16#4328 THEN
		stErrorMessage := 'Loop movement not allowed';
	END_IF
	IF NC_Error_Code = 16#4329 THEN
		stErrorMessage := 'Axis cycle time not allowed';
	END_IF
	IF NC_Error_Code = 16#432E THEN
		stErrorMessage := 'DWORD for the interpretation of the axis units not allowed';
	END_IF
	IF NC_Error_Code = 16#432F THEN
		stErrorMessage := 'Maximum velocity not allowed';
	END_IF
	IF NC_Error_Code = 16#4330 THEN
		stErrorMessage := 'Motion monitoring window not allowed';
	END_IF
	IF NC_Error_Code = 16#4331 THEN
		stErrorMessage := 'PEH time monitoring not allowed';
	END_IF
	IF NC_Error_Code = 16#4332 THEN
		stErrorMessage := 'PEH monitoring time not allowed';
	END_IF
	IF NC_Error_Code = 16#4333 THEN
		stErrorMessage := 'AXISERR_RANGE_DELAYBREAKRELEASE';
	END_IF
	IF NC_Error_Code = 16#4334 THEN
		stErrorMessage := 'AXISERR_RANGE_DATAPERSISTENCE';
	END_IF
	IF NC_Error_Code = 16#4340 THEN
		stErrorMessage := 'Axis initialisation';
	END_IF
	IF NC_Error_Code = 16#4342 THEN
		stErrorMessage := 'Encoder address';
	END_IF
	IF NC_Error_Code = 16#4343 THEN
		stErrorMessage := 'Controller address';
	END_IF
	IF NC_Error_Code = 16#4344 THEN
		stErrorMessage := 'Drive address';
	END_IF
	IF NC_Error_Code = 16#4345 THEN
		stErrorMessage := 'Axis interface PLC to NC address';
	END_IF
	IF NC_Error_Code = 16#4346 THEN
		stErrorMessage := 'Axis interface NC to PLC address';
	END_IF
	IF NC_Error_Code = 16#4356 THEN
		stErrorMessage := 'Controller enable';
	END_IF
	IF NC_Error_Code = 16#4357 THEN
		stErrorMessage := 'Feed enable minus';
	END_IF
	IF NC_Error_Code = 16#4358 THEN
		stErrorMessage := 'Feed enable plus';
	END_IF
	IF NC_Error_Code = 16#4359 THEN
		stErrorMessage := 'Set velocity not allowed';
	END_IF
	IF NC_Error_Code = 16#435A THEN
		stErrorMessage := 'Movement smaller than one encoder increment';
	END_IF
	IF NC_Error_Code = 16#435B THEN
		stErrorMessage := 'Set acceleration monitoring';
	END_IF
	IF NC_Error_Code = 16#435C THEN
		stErrorMessage := 'PEH time monitoring';
	END_IF
	IF NC_Error_Code = 16#435D THEN
		stErrorMessage := 'Encoder existence monitoring / movement monitoring';
	END_IF
	IF NC_Error_Code = 16#435E THEN
		stErrorMessage := 'Looping distance less than breaking distance';
	END_IF
	IF NC_Error_Code = 16#43A0 THEN
		stErrorMessage := 'Axis consequential error';
	END_IF
END_IF


(*Encoder Errors*)
IF dwMask = 16#44 THEN
	stGroupMessage := 'Encoder Error: ';
	IF NC_Error_Code = 16#4402 THEN
		stErrorMessage := 'Encoder mode';
	END_IF
	IF NC_Error_Code = 16#4403 THEN
		stErrorMessage := 'Encoder counting direction inverted?';
	END_IF
	IF NC_Error_Code = 16#4404 THEN
		stErrorMessage := 'Referencing status';
	END_IF
	IF NC_Error_Code = 16#4405 THEN
		stErrorMessage := 'Encoder increments for each physical encoder rotation';
	END_IF
	IF NC_Error_Code = 16#4406 THEN
		stErrorMessage := 'Scaling factor';
	END_IF
	IF NC_Error_Code = 16#4407 THEN
		stErrorMessage := 'Position offset (zero point offset)';
	END_IF
	IF NC_Error_Code = 16#4408 THEN
		stErrorMessage := 'Modulo factor';
	END_IF
	IF NC_Error_Code = 16#4409 THEN
		stErrorMessage := 'Position filter time';
	END_IF
	IF NC_Error_Code = 16#440A THEN
		stErrorMessage := 'Velocity filter time';
	END_IF
	IF NC_Error_Code = 16#440B THEN
		stErrorMessage := 'Acceleration filter time';
	END_IF
	IF NC_Error_Code = 16#440C THEN
		stErrorMessage := 'Cycle time not allowed';
	END_IF
	IF NC_Error_Code = 16#440E THEN
		stErrorMessage := 'Actual position correction / measurement system error correction';
	END_IF
	IF NC_Error_Code = 16#440F THEN
		stErrorMessage := 'Filter time actual position correction';
	END_IF
	IF NC_Error_Code = 16#4410 THEN
		stErrorMessage := 'Search direction for referencing cam inverted';
	END_IF
	IF NC_Error_Code = 16#4411 THEN
		stErrorMessage := 'Search direction for sync pulse (zero pulse) inverted';
	END_IF
	IF NC_Error_Code = 16#4412 THEN
		stErrorMessage := 'Reference position';
	END_IF
	IF NC_Error_Code = 16#4413 THEN
		stErrorMessage := 'Clearance monitoring between activation of the hardware latch and appearance of the sync pulse" (NOT IMPLEMENTED)';
	END_IF
	IF NC_Error_Code = 16#4414 THEN
		stErrorMessage := 'Minimum clearance between activation of the hardware latch and appearance of the sync pulse" (NOT IMPLEMENTED)';
	END_IF
	IF NC_Error_Code = 16#4415 THEN
		stErrorMessage := 'External sync pulse" (NOT IMPLEMENTED)';
	END_IF
	IF NC_Error_Code = 16#4416 THEN
		stErrorMessage := 'Scaling of the noise rate is not allowed';
	END_IF
	IF NC_Error_Code = 16#4417 THEN
		stErrorMessage := 'Tolerance window for modulo-start';
	END_IF
	IF NC_Error_Code = 16#4418 THEN
		stErrorMessage := 'Encoder reference mode';
	END_IF
	IF NC_Error_Code = 16#4419 THEN
		stErrorMessage := 'Encoder evaluation direction';
	END_IF
	IF NC_Error_Code = 16#441A THEN
		stErrorMessage := 'Encoder reference system';
	END_IF
	IF NC_Error_Code = 16#441B THEN
		stErrorMessage := 'Encoder position initialization mode';
	END_IF
	IF NC_Error_Code = 16#441C THEN
		stErrorMessage := 'Encoder sign interpretation (UNSIGNED- / SIGNED- data type)“';
	END_IF
	IF NC_Error_Code = 16#4420 THEN
		stErrorMessage := 'Software end location monitoring minimum not allowed';
	END_IF
	IF NC_Error_Code = 16#4421 THEN
		stErrorMessage := 'Software end location monitoring maximum not allowed';
	END_IF
	IF NC_Error_Code = 16#4422 THEN
		stErrorMessage := 'Actual value setting is outside the value range';
	END_IF
	IF NC_Error_Code = 16#4423 THEN
		stErrorMessage := 'Software end location minimum not allowed';
	END_IF
	IF NC_Error_Code = 16#4424 THEN
		stErrorMessage := 'Software end location maximum not allowed';
	END_IF
	IF NC_Error_Code = 16#4425 THEN
		stErrorMessage := 'Filter mask for the raw data of the encoder is invalid';
	END_IF
	IF NC_Error_Code = 16#4426 THEN
		stErrorMessage := 'Reference mask for the raw data of the encoder is invalid';
	END_IF
	IF NC_Error_Code = 16#4430 THEN
		stErrorMessage := 'Hardware latch activation (encoder)';
	END_IF
	IF NC_Error_Code = 16#4431 THEN
		stErrorMessage := 'External hardware latch activation (encoder)';
	END_IF
	IF NC_Error_Code = 16#4432 THEN
		stErrorMessage := 'External hardware latch activation (encoder)';
	END_IF
	IF NC_Error_Code = 16#4433 THEN
		stErrorMessage := 'External hardware latch activation (encoder)';
	END_IF
	IF NC_Error_Code = 16#4434 THEN
		stErrorMessage := 'Encoder function not supported';
	END_IF
	IF NC_Error_Code = 16#4435 THEN
		stErrorMessage := 'Encoder function is already active';
	END_IF
	IF NC_Error_Code = 16#4440 THEN
		stErrorMessage := 'Encoder initialization';
	END_IF
	IF NC_Error_Code = 16#4441 THEN
		stErrorMessage := 'Axis address';
	END_IF
	IF NC_Error_Code = 16#4442 THEN
		stErrorMessage := 'I/O input structure address';
	END_IF
	IF NC_Error_Code = 16#4443 THEN
		stErrorMessage := 'I/O output structure address';
	END_IF
	IF NC_Error_Code = 16#4450 THEN
		stErrorMessage := 'Encoder counter underflow monitoring';
	END_IF
	IF NC_Error_Code = 16#4451 THEN
		stErrorMessage := 'Encoder counter overflow monitoring';
	END_IF
	IF NC_Error_Code = 16#4460 THEN
		stErrorMessage := 'Software end location minimum (axis start)';
	END_IF
	IF NC_Error_Code = 16#4461 THEN
		stErrorMessage := 'Software end location maximum (axis start)';
	END_IF
	IF NC_Error_Code = 16#4462 THEN
		stErrorMessage := 'Software end location minimum (positioning process)" ';
	END_IF
	IF NC_Error_Code = 16#4463 THEN
		stErrorMessage := 'Software end location maximum (positioning process)';
	END_IF
	IF NC_Error_Code = 16#4464 THEN
		stErrorMessage := 'Encoder hardware error';
	END_IF
	IF NC_Error_Code = 16#4465 THEN
		stErrorMessage := 'Position initialization error at system start';
	END_IF
	IF NC_Error_Code = 16#4470 THEN
		stErrorMessage := 'SSI transformation fault or not finished';
	END_IF
	IF NC_Error_Code = 16#44A2 THEN
		stErrorMessage := 'ENCERR_ADDR_CONTROLLER';
	END_IF
	IF NC_Error_Code = 16#44A3 THEN
		stErrorMessage := 'ENCERR_INVALID_CONTROLLERTYPE';
	END_IF
END_IF

(*Controller Errors*)
IF dwMask = 16#45 THEN
	stGroupMessage := 'Controller Error: ';
	IF NC_Error_Code = 16#4500 THEN
		stErrorMessage := 'Controller ID not allowed';
	END_IF
	IF NC_Error_Code = 16#4501 THEN
		stErrorMessage := 'Controller type not allowed';
	END_IF
	IF NC_Error_Code = 16#4502 THEN
		stErrorMessage := 'Controller operating mode not allowed';
	END_IF
	IF NC_Error_Code = 16#4503 THEN
		stErrorMessage := 'Weighting of the velocity pre-control not allowed';
	END_IF
	IF NC_Error_Code = 16#4504 THEN
		stErrorMessage := 'Following error monitoring (position) not allowed';
	END_IF
	IF NC_Error_Code = 16#4505 THEN
		stErrorMessage := 'Following error (velocity) not allowed';
	END_IF
	IF NC_Error_Code = 16#4506 THEN
		stErrorMessage := 'Following error window (position) not allowed';
	END_IF
	IF NC_Error_Code = 16#4507 THEN
		stErrorMessage := 'Following error filter time (position) not allowed';
	END_IF
	IF NC_Error_Code = 16#4508 THEN
		stErrorMessage := 'Following error window (velocity) not allowed';
	END_IF
	IF NC_Error_Code = 16#4509 THEN
		stErrorMessage := 'Following error filter time (velocity) not allowed';
	END_IF
	IF NC_Error_Code = 16#4510 THEN
		stErrorMessage := 'Proportional gain Kv or Kp (position controller) not allowed';
	END_IF
	IF NC_Error_Code = 16#4511 THEN
		stErrorMessage := 'Integral-action time Tn (position controller) not allowed';
	END_IF
	IF NC_Error_Code = 16#4512 THEN
		stErrorMessage := 'Derivative action time Tv (position controller) not allowed';
	END_IF
	IF NC_Error_Code = 16#4513 THEN
		stErrorMessage := 'Damping time Td (position controller) not allowed';
	END_IF
	IF NC_Error_Code = 16#4514 THEN
		stErrorMessage := 'Activation of the automatic offset compensation not allowed';
	END_IF
	IF NC_Error_Code = 16#4515 THEN
		stErrorMessage := 'Additional proportional gain Kv or Kp (position controller) not allowed';
	END_IF
	IF NC_Error_Code = 16#4516 THEN
		stErrorMessage := 'Reference velocity for additional proportional gain Kv or Kp (position controller) not allowed';
	END_IF
	IF NC_Error_Code = 16#4517 THEN
		stErrorMessage := 'Proportional gain Pa (acceleration proportion) not allowed';
	END_IF
	IF NC_Error_Code = 16#4518 THEN
		stErrorMessage := 'Proportional gain Kv (velocity controller) not allowed';
	END_IF
	IF NC_Error_Code = 16#4519 THEN
		stErrorMessage := 'Reset time Tn (velocity controller) not allowed';
	END_IF
	IF NC_Error_Code = 16#451A THEN
		stErrorMessage := 'CONTROLERR_RANGE_ACCJUMPLIMITINGMODE';
	END_IF
	IF NC_Error_Code = 16#451B THEN
		stErrorMessage := 'CONTROLERR_RANGE_ACCJUMPVALUE';
	END_IF
	IF NC_Error_Code = 16#451C THEN
		stErrorMessage := 'CONTROLERR_RANGE_FILTERTIME';
	END_IF
	IF NC_Error_Code = 16#451D THEN
		stErrorMessage := 'Dead zone not allowed';
	END_IF
	IF NC_Error_Code = 16#4520 THEN
		stErrorMessage := 'Rate time Tv (velocity controller) not allowed';
	END_IF
	IF NC_Error_Code = 16#4521 THEN
		stErrorMessage := 'Damping time Td (velocity controller) not allowed';
	END_IF
	IF NC_Error_Code = 16#4522 THEN
		stErrorMessage := 'CONTROLERR_RANGE_IOUTPUTLIMIT';
	END_IF
	IF NC_Error_Code = 16#4523 THEN
		stErrorMessage := 'CONTROLERR_RANGE_DOUTPUTLIMIT';
	END_IF
	IF NC_Error_Code = 16#4524 THEN
		stErrorMessage := 'CONTROLERR_RANGE_POSIDISABLEWHENMOVING';
	END_IF
	IF NC_Error_Code = 16#4540 THEN
		stErrorMessage := 'Controller initialisation';
	END_IF
	IF NC_Error_Code = 16#4541 THEN
		stErrorMessage := 'Axis address';
	END_IF
	IF NC_Error_Code = 16#4542 THEN
		stErrorMessage := 'Drive address';
	END_IF
	IF NC_Error_Code = 16#4550 THEN
		stErrorMessage := 'Following error monitoring (position)';
	END_IF
	IF NC_Error_Code = 16#4551 THEN
		stErrorMessage := 'Following error monitoring (velocity)';
	END_IF
	IF NC_Error_Code = 16#45A0 THEN
		stErrorMessage := 'CONTROLERR_RANGE_AREA_ASIDE';
	END_IF
	IF NC_Error_Code = 16#45A1 THEN
		stErrorMessage := 'CONTROLERR_RANGE_AREA_BSIDE';
	END_IF
	IF NC_Error_Code = 16#45A2 THEN
		stErrorMessage := 'CONTROLERR_RANGE_QNENN';
	END_IF
	IF NC_Error_Code = 16#45A3 THEN
		stErrorMessage := 'CONTROLERR_RANGE_PNENN';
	END_IF
	IF NC_Error_Code = 16#45A4 THEN
		stErrorMessage := 'CONTROLERR_RANGE_AXISIDPRESP0';
	END_IF
END_IF

(*Drive Error*)
IF dwMask = 16#46 THEN
	stGroupMessage := 'Drive Error: ';
	IF NC_Error_Code = 16#4600 THEN
		stErrorMessage := 'Drive ID not allowed';
	END_IF
	IF NC_Error_Code = 16#4601 THEN
		stErrorMessage := 'Drive type not allowed';
	END_IF
	IF NC_Error_Code = 16#4602 THEN
		stErrorMessage := 'Drive operating mode not allowed';
	END_IF
	IF NC_Error_Code = 16#4603 THEN
		stErrorMessage := 'Motor polarity inverted?';
	END_IF
	IF NC_Error_Code = 16#4604 THEN
		stErrorMessage := 'Drift compensation/velocity offset (DAC offset)';
	END_IF
	IF NC_Error_Code = 16#4605 THEN
		stErrorMessage := 'Reference velocity (velocity pre-control)';
	END_IF
	IF NC_Error_Code = 16#4606 THEN
		stErrorMessage := 'Reference output in percent';
	END_IF
	IF NC_Error_Code = 16#4607 THEN
		stErrorMessage := 'Quadrant compensation factor';
	END_IF
	IF NC_Error_Code = 16#4608 THEN
		stErrorMessage := 'Velocity reference point in percent';
	END_IF
	IF NC_Error_Code = 16#4609 THEN
		stErrorMessage := 'Output reference point in percent';
	END_IF
	IF NC_Error_Code = 16#460A THEN
		stErrorMessage := 'Minimum or maximum output limit';
	END_IF
	IF NC_Error_Code = 16#460B THEN
		stErrorMessage := 'DRIVEERR_RANGE_MAXINCREMENT';
	END_IF
	IF NC_Error_Code = 16#460C THEN
		stErrorMessage := 'DRIVEERR_RANGE_ DRIVECONTROLDWORD';
	END_IF
	IF NC_Error_Code = 16#460D THEN
		stErrorMessage := 'DRIVEERR_RANGE_ RESETCYCLECOUNTER';
	END_IF
	IF NC_Error_Code = 16#460F THEN
		stErrorMessage := 'Drive torque output scaling is not allowed';
	END_IF
	IF NC_Error_Code = 16#4610 THEN
		stErrorMessage := 'Drive velocity output scaling is not allowed';
	END_IF
	IF NC_Error_Code = 16#4611 THEN
		stErrorMessage := 'Profi Drive DSC Proportional gain  Kpc (position controller) not allowed';
	END_IF
	IF NC_Error_Code = 16#4612 THEN
		stErrorMessage := 'Table-ID is invalid';
	END_IF
	IF NC_Error_Code = 16#4613 THEN
		stErrorMessage := 'Table interpolationtype is invalid';
	END_IF
	IF NC_Error_Code = 16#4614 THEN
		stErrorMessage := 'Outputoffset in percent is invalid';
	END_IF
	IF NC_Error_Code = 16#4615 THEN
		stErrorMessage := 'Profi Drive DSC scaling factor for calculating Xerr (position controller) is not allowed';
	END_IF
	IF NC_Error_Code = 16#4616 THEN
		stErrorMessage := 'Drive acceleration output scaling is not allowed';
	END_IF
	IF NC_Error_Code = 16#4617 THEN
		stErrorMessage := 'Drive position output scaling is not allowed';
	END_IF
	IF NC_Error_Code = 16#4620 THEN
		stErrorMessage := 'Bit mask for stepper motor cycle not allowed';
	END_IF
	IF NC_Error_Code = 16#4621 THEN
		stErrorMessage := 'Bit mask for stepper motor holding current not allowed';
	END_IF
	IF NC_Error_Code = 16#4640 THEN
		stErrorMessage := 'Drive initialisation';
	END_IF
	IF NC_Error_Code = 16#4641 THEN
		stErrorMessage := 'Axis address';
	END_IF
	IF NC_Error_Code = 16#4642 THEN
		stErrorMessage := 'I/O input structure address';
	END_IF
	IF NC_Error_Code = 16#4643 THEN
		stErrorMessage := 'I/O output structure address';
	END_IF
	IF NC_Error_Code = 16#4650 THEN
		stErrorMessage := 'Drive not ready for operation';
	END_IF
	IF NC_Error_Code = 16#4651 THEN
		stErrorMessage := 'Error in cyclic communication with the drive (life counter)';
	END_IF
	IF NC_Error_Code = 16#4652 THEN
		stErrorMessage := 'Not permitted to change the table ID while the axis is enabled';
	END_IF
	IF NC_Error_Code = 16#4655 THEN
		stErrorMessage := 'Invalid IO data for more than (n) consecutive nc cycles';
	END_IF
END_IF

